(* IEC 61131-3 sources: verifaps-lib/share/PPU.stold (part 6) *)

(* ---- Scenario13_Final.xml.st ---- *)
TYPE
    Crane_states_t : (Crane_Go_Up , Crane_Go_Up_White , Crane_Init , Crane_Init_2 , Crane_Lift_At_Stamp , Crane_Lift_At_Stamp2 , Crane_Lift_Conveyor , Crane_Lift_Conveyor2 , Crane_Lift_Conveyor_Black , Crane_Lift_Magazin , Crane_Lift_Magazin_Metallic , Crane_Lift_Magazin_White , Crane_Lift_NOT_Metallic_Black , Crane_Lower , Crane_On_Conveyor , Crane_On_Conveyor_Metallic , Crane_On_Conveyor_Metallic2 , Crane_On_Conveyor_Not_Metallica_Black , Crane_On_Stamp_Metallic , Crane_On_Stamp_Metallic2 , Crane_On_Stamp_Metallic2_Lower , Crane_On_Stamp_Stop_Black , Crane_On_Stamp_White , Crane_Turn_Left_Back_To_Stamp , Crane_Turn_Left_From_Stamp , Crane_Turn_Left_Metallic , Crane_Turn_Left_Metallic2 , Crane_Turn_Left_NOT_Metallic , Crane_Turn_Left_NOT_Metallic_Black , Crane_Turn_Left_White , Crane_Turn_Right_From_Stamp , Init , Interstep , Interstep_2 , Interstep_3 , Interstep_4 , Lower_Crane , Magazin_Stop , Magazin_Stop_Black , Magazin_Stop_Final , No_Workpiece_ready , Reset_interconnect , Stamp_Pressure_Profile_Set_Metallic , Stamp_Pressure_Profile_Set_White , Start_Crane , Step0 , Step2 , Step3 , Step4 , Suck_At_Stamp , Suck_At_Stamp2 , TimeDelay , Turn_Right , Turn_Right_Black , Turn_Right_Final , pause , release , release2 , release_Black , release_Workpiece , release_Workpiece_White);
    Magazin_states_t : (Green_Lamp , Init , Interstep , Magazin_Init , Magazin_Init_2 , Slider_Move_Back , Start_Magazin , Step0 , Step1 , convey);
    Conveyor_states_t : (Conveyor_Init , Conveyor_Stop_Empty_Magazin , Conveyor_Towards_Stacker , Conveyor_init_2 , Conveyor_pause , Green_Lamp , Init , Interstep , Runtime_Conveyor , Start_Conveyor , Step0);
    Stamp_states_t : (Green_Lamp , Init , Interstep , Intertsep_2 , StampProcess , StampSliderBack , StampSliderForward , Stamp_Init_1 , Stamp_Init_2 , Stamp_Init_3 , Stamp_Init_4 , Start_Stamp , Step0 , Step1 , Step2);
    Pusher_states_t : (Check_For_Black , Check_For_Metal , Check_For_White , First_Slide_Timer_Black , First_Slide_Timer_Metal , First_Slide_Timer_White , First_Slide_black_workpieces , First_Slide_metal_workpieces , First_Slide_white_workpieces , Init , Interstep , Interstep_2 , PusherY1_Move_In_Black , PusherY1_Move_In_Metal , PusherY1_Move_In_White , PusherY1_Move_Out_Black , PusherY1_Move_Out_Metal , PusherY1_Move_Out_White , PusherY2_Move_In_Black , PusherY2_Move_In_Metal , PusherY2_Move_In_White , PusherY2_Move_Out_Black , PusherY2_Move_Out_Metal , PusherY2_Move_Out_White , Reset_interconnect3 , Reset_interconnect_Slide1_Black , Reset_interconnect_Slide1_Metal , Reset_interconnect_Slide1_White , Reset_interconnect_Slide2_Black , Reset_interconnect_Slide2_Metal , Reset_interconnect_Slide2_White , Reset_interconnect_Slide3_Metal , Reset_interconnect_Slide3_White , Second_Slide_Timer_Black , Second_Slide_Timer_Metal , Second_Slide_Timer_White , Second_Slide_black_workpieces , Second_Slide_metal_workpieces , Second_Slide_white_workpieces , Second_Test_For_Metal , Second_Test_For_White , Third_Slide_black_workpieces , Third_Slide_metal_workpieces , Third_Slide_white_workpieces , Wait_Black , Wait_Metal , Wait_White , Wait_Y1_Black , Wait_Y1_Metal , Wait_Y1_White , Wait_Y2_Black , Wait_Y2_Metal , Wait_Y2_White);
END_TYPE

FUNCTION_BLOCK Crane
    VAR_INPUT  AnalogCranePosition : INT; END_VAR {*Irwxp*}
    VAR_OUTPUT  AnalogCranePressure : INT; END_VAR {*Orwxp*}
    VAR_INPUT  CraneDown : BOOL; END_VAR {*Irwxp*}
    VAR_OUTPUT  CraneLower : BOOL; END_VAR {*Orwxp*}
    VAR_INPUT  CraneSucked : BOOL; END_VAR {*Irwxp*}
    VAR_OUTPUT  CraneTurnClockwise : BOOL; END_VAR {*Orwxp*}
    VAR_OUTPUT  CraneTurnCounterclockwise : BOOL; END_VAR {*Orwxp*}
    VAR_INPUT  CraneUp : BOOL; END_VAR {*Irwxp*}
    VAR  Duration1 : TIME := TIME#1.0s500.0ms; END_VAR {*Lrwxp*}
    VAR_INPUT  MagazinCapacitiveSensor : BOOL; END_VAR {*Irwxp*}
    VAR_INPUT  MagazinOpticalSensor : BOOL; END_VAR {*Irwxp*}
    VAR_OUTPUT  MagazinSlider : BOOL; END_VAR {*Orwxp*}
    VAR_OUTPUT  MagazinVacuumOff : BOOL; END_VAR {*Orwxp*}
    VAR_OUTPUT  MagazinVacuumOn : BOOL; END_VAR {*Orwxp*}
    VAR  SFCInit : BOOL; END_VAR {*Lrwxp*}
    VAR_INPUT  SFCReset : BOOL; END_VAR {*Irwxp*}
    VAR_INPUT  SliderMovedOut : BOOL; END_VAR {*Irwxp*}
    VAR_INPUT  SliderNotMovedOut : BOOL; END_VAR {*Irwxp*}
    VAR_INPUT  StampLowered : BOOL; END_VAR {*Irwxp*}
    VAR_INPUT  StampSliderFilled : BOOL; END_VAR {*Irwxp*}
    VAR_INPUT  StampSliderSensorMovedOut : BOOL; END_VAR {*Irwxp*}
    VAR_INPUT  StartButtonMagazin : BOOL; END_VAR {*Irwxp*}
    VAR_OUTPUT  StartCommandCrane : BOOL; END_VAR {*Orwxp*}
    VAR_INPUT  StartVar : BOOL; END_VAR {*Irwxp*}
    VAR  TimeDelay_Timer : TON; END_VAR {*Lrwxp*}
    VAR  TimeDelay_Timer_Duration : TIME := TIME#50.0ms; END_VAR {*Lrwxp*}
    VAR  TimeDelay_Timer_interconnect : BOOL; END_VAR {*Lrwxp*}
    VAR  Timer1 : TON; END_VAR {*Lrwxp*}
    VAR_INPUT  WorkpieceReady : BOOL; END_VAR {*Irwxp*}
    VAR  _state : Crane_states_t; END_VAR {*Lrwxp*}
    VAR  _transit : BOOL; END_VAR {*Lrwxp*}
    VAR  actualtime1 : TIME; END_VAR {*Lrwxp*}
    VAR  interconnect : BOOL; END_VAR {*Lrwxp*}
    VAR  interconnectCraneStartCommand : BOOL; END_VAR {*Lrwxp*}

    CASE _state OF
        Crane_states_t#Crane_Go_Up:
            {* begin(State) *}
            {* begin(onEntry) *}
            _transit := FALSE;
            {* end(onEntry) *}
            {* begin(onActive) *}
            CraneLower := FALSE;
            {* end(onActive) *}
            {* begin(transition) *}
            IF CraneUp THEN
                _transit := TRUE;
                _state := Crane_states_t#Step3;
            END_IF;
            {* end(transition) *}
            {* begin(onExit) *}
            {* end(onExit) *}
            {* end(State) *}

        Crane_states_t#Crane_Go_Up_White:
            {* begin(State) *}
            {* begin(onEntry) *}
            _transit := FALSE;
            {* end(onEntry) *}
            {* begin(onActive) *}
            CraneLower := FALSE;
            {* end(onActive) *}
            {* begin(transition) *}
            IF CraneUp THEN
                _transit := TRUE;
                _state := Crane_states_t#Step3;
            END_IF;
            {* end(transition) *}
            {* begin(onExit) *}
            {* end(onExit) *}
            {* end(State) *}

        Crane_states_t#Crane_Init:
            {* begin(State) *}
            {* begin(onEntry) *}
            _transit := FALSE;
            {* end(onEntry) *}
            {* begin(onActive) *}
            CraneLower := TRUE;
            interconnectCraneStartCommand := FALSE;
            AnalogCranePressure := INT#6000;
            {* end(onActive) *}
            {* begin(transition) *}
            IF CraneDown THEN
                _transit := TRUE;
                _state := Crane_states_t#Crane_Init_2;
            END_IF;
            {* end(transition) *}
            {* begin(onExit) *}
            {* end(onExit) *}
            {* end(State) *}

        Crane_states_t#Crane_Init_2:
            {* begin(State) *}
            {* begin(onEntry) *}
            _transit := FALSE;
            {* end(onEntry) *}
            {* begin(onActive) *}
            CraneLower := FALSE;
            {* end(onActive) *}
            {* begin(transition) *}
            IF CraneUp THEN
                _transit := TRUE;
                _state := Crane_states_t#Interstep;
            END_IF;
            {* end(transition) *}
            {* begin(onExit) *}
            {* end(onExit) *}
            {* end(State) *}

        Crane_states_t#Crane_Lift_At_Stamp:
            {* begin(State) *}
            {* begin(onEntry) *}
            _transit := FALSE;
            {* end(onEntry) *}
            {* begin(onActive) *}
            CraneLower := FALSE;
            {* end(onActive) *}
            {* begin(transition) *}
            IF CraneUp THEN
                _transit := TRUE;
                _state := Crane_states_t#Crane_Turn_Left_From_Stamp;
            END_IF;
            {* end(transition) *}
            {* begin(onExit) *}
            {* end(onExit) *}
            {* end(State) *}

        Crane_states_t#Crane_Lift_At_Stamp2:
            {* begin(State) *}
            {* begin(onEntry) *}
            _transit := FALSE;
            {* end(onEntry) *}
            {* begin(onActive) *}
            CraneLower := FALSE;
            AnalogCranePressure := INT#0;
            {* end(onActive) *}
            {* begin(transition) *}
            IF CraneUp THEN
                _transit := TRUE;
                _state := Crane_states_t#Crane_Turn_Right_From_Stamp;
            END_IF;
            {* end(transition) *}
            {* begin(onExit) *}
            {* end(onExit) *}
            {* end(State) *}

        Crane_states_t#Crane_Lift_Conveyor:
            {* begin(State) *}
            {* begin(onEntry) *}
            _transit := FALSE;
            {* end(onEntry) *}
            {* begin(onActive) *}
            CraneLower := FALSE;
            {* end(onActive) *}
            {* begin(transition) *}
            IF TRUE THEN
                _transit := TRUE;
                _state := Crane_states_t#Interstep;
            END_IF;
            {* end(transition) *}
            {* begin(onExit) *}
            {* end(onExit) *}
            {* end(State) *}

        Crane_states_t#Crane_Lift_Conveyor2:
            {* begin(State) *}
            {* begin(onEntry) *}
            _transit := FALSE;
            {* end(onEntry) *}
            {* begin(onActive) *}
            CraneLower := FALSE;
            {* end(onActive) *}
            {* begin(transition) *}
            IF TRUE THEN
                _transit := TRUE;
                _state := Crane_states_t#Interstep;
            END_IF;
            {* end(transition) *}
            {* begin(onExit) *}
            {* end(onExit) *}
            {* end(State) *}

        Crane_states_t#Crane_Lift_Conveyor_Black:
            {* begin(State) *}
            {* begin(onEntry) *}
            _transit := FALSE;
            {* end(onEntry) *}
            {* begin(onActive) *}
            CraneLower := FALSE;
            {* end(onActive) *}
            {* begin(transition) *}
            IF CraneUp THEN
                _transit := TRUE;
                _state := Crane_states_t#Crane_Turn_Left_Back_To_Stamp;
            END_IF;
            {* end(transition) *}
            {* begin(onExit) *}
            {* end(onExit) *}
            {* end(State) *}

        Crane_states_t#Crane_Lift_Magazin:
            {* begin(State) *}
            {* begin(onEntry) *}
            _transit := FALSE;
            {* end(onEntry) *}
            {* begin(onActive) *}
            CraneLower := FALSE;
            {* end(onActive) *}
            {* begin(transition) *}
            IF CraneUp THEN
                _transit := TRUE;
                _state := Crane_states_t#Crane_Turn_Left_NOT_Metallic;
            END_IF;
            {* end(transition) *}
            {* begin(onExit) *}
            {* end(onExit) *}
            {* end(State) *}

        Crane_states_t#Crane_Lift_Magazin_Metallic:
            {* begin(State) *}
            {* begin(onEntry) *}
            _transit := FALSE;
            {* end(onEntry) *}
            {* begin(onActive) *}
            CraneLower := FALSE;
            {* end(onActive) *}
            {* begin(transition) *}
            IF CraneUp THEN
                _transit := TRUE;
                _state := Crane_states_t#Crane_Turn_Left_Metallic;
            END_IF;
            {* end(transition) *}
            {* begin(onExit) *}
            {* end(onExit) *}
            {* end(State) *}

        Crane_states_t#Crane_Lift_Magazin_White:
            {* begin(State) *}
            {* begin(onEntry) *}
            _transit := FALSE;
            {* end(onEntry) *}
            {* begin(onActive) *}
            CraneLower := FALSE;
            {* end(onActive) *}
            {* begin(transition) *}
            IF CraneUp THEN
                _transit := TRUE;
                _state := Crane_states_t#Crane_Turn_Left_White;
            END_IF;
            {* end(transition) *}
            {* begin(onExit) *}
            {* end(onExit) *}
            {* end(State) *}

        Crane_states_t#Crane_Lift_NOT_Metallic_Black:
            {* begin(State) *}
            {* begin(onEntry) *}
            _transit := FALSE;
            {* end(onEntry) *}
            {* begin(onActive) *}
            CraneLower := FALSE;
            {* end(onActive) *}
            {* begin(transition) *}
            IF CraneUp THEN
                _transit := TRUE;
                _state := Crane_states_t#Crane_Turn_Left_NOT_Metallic_Black;
            END_IF;
            {* end(transition) *}
            {* begin(onExit) *}
            {* end(onExit) *}
            {* end(State) *}

        Crane_states_t#Crane_Lower:
            {* begin(State) *}
            {* begin(onEntry) *}
            _transit := FALSE;
            {* end(onEntry) *}
            {* begin(onActive) *}
            MagazinVacuumOn := TRUE;
            MagazinVacuumOff := FALSE;
            CraneLower := TRUE;
            AnalogCranePressure := INT#0;
            {* end(onActive) *}
            {* begin(transition) *}
            IF CraneSucked THEN
                _transit := TRUE;
                _state := Crane_states_t#Step0;
            END_IF;
            {* end(transition) *}
            {* begin(onExit) *}
            {* end(onExit) *}
            {* end(State) *}

        Crane_states_t#Crane_On_Conveyor:
            {* begin(State) *}
            {* begin(onEntry) *}
            _transit := FALSE;
            {* end(onEntry) *}
            {* begin(onActive) *}
            CraneTurnCounterclockwise := FALSE;
            CraneTurnClockwise := FALSE;
            CraneLower := TRUE;
            {* end(onActive) *}
            {* begin(transition) *}
            IF CraneDown THEN
                _transit := TRUE;
                _state := Crane_states_t#release;
            END_IF;
            {* end(transition) *}
            {* begin(onExit) *}
            {* end(onExit) *}
            {* end(State) *}

        Crane_states_t#Crane_On_Conveyor_Metallic:
            {* begin(State) *}
            {* begin(onEntry) *}
            _transit := FALSE;
            {* end(onEntry) *}
            {* begin(onActive) *}
            CraneTurnCounterclockwise := FALSE;
            CraneTurnClockwise := FALSE;
            CraneLower := TRUE;
            {* end(onActive) *}
            {* begin(transition) *}
            IF CraneDown THEN
                _transit := TRUE;
                _state := Crane_states_t#release;
            END_IF;
            {* end(transition) *}
            {* begin(onExit) *}
            {* end(onExit) *}
            {* end(State) *}

        Crane_states_t#Crane_On_Conveyor_Metallic2:
            {* begin(State) *}
            {* begin(onEntry) *}
            _transit := FALSE;
            {* end(onEntry) *}
            {* begin(onActive) *}
            CraneTurnCounterclockwise := FALSE;
            CraneTurnClockwise := FALSE;
            CraneLower := TRUE;
            {* end(onActive) *}
            {* begin(transition) *}
            IF CraneDown THEN
                _transit := TRUE;
                _state := Crane_states_t#release2;
            END_IF;
            {* end(transition) *}
            {* begin(onExit) *}
            {* end(onExit) *}
            {* end(State) *}

        Crane_states_t#Crane_On_Conveyor_Not_Metallica_Black:
            {* begin(State) *}
            {* begin(onEntry) *}
            _transit := FALSE;
            {* end(onEntry) *}
            {* begin(onActive) *}
            CraneTurnCounterclockwise := FALSE;
            CraneTurnClockwise := FALSE;
            CraneLower := TRUE;
            {* end(onActive) *}
            {* begin(transition) *}
            IF CraneDown THEN
                _transit := TRUE;
                _state := Crane_states_t#release_Black;
            END_IF;
            {* end(transition) *}
            {* begin(onExit) *}
            {* end(onExit) *}
            {* end(State) *}

        Crane_states_t#Crane_On_Stamp_Metallic:
            {* begin(State) *}
            {* begin(onEntry) *}
            _transit := FALSE;
            {* end(onEntry) *}
            {* begin(onActive) *}
            CraneTurnCounterclockwise := FALSE;
            CraneTurnClockwise := FALSE;
            CraneLower := TRUE;
            {* end(onActive) *}
            {* begin(transition) *}
            IF CraneDown THEN
                _transit := TRUE;
                _state := Crane_states_t#release_Workpiece;
            END_IF;
            {* end(transition) *}
            {* begin(onExit) *}
            {* end(onExit) *}
            {* end(State) *}

        Crane_states_t#Crane_On_Stamp_Metallic2:
            {* begin(State) *}
            {* begin(onEntry) *}
            _transit := FALSE;
            {* end(onEntry) *}
            {* begin(onActive) *}
            CraneTurnCounterclockwise := FALSE;
            CraneTurnClockwise := FALSE;
            {* end(onActive) *}
            {* begin(transition) *}
            IF StampLowered THEN
                _transit := TRUE;
                _state := Crane_states_t#Interstep_4;
            END_IF;
            {* end(transition) *}
            {* begin(onExit) *}
            {* end(onExit) *}
            {* end(State) *}

        Crane_states_t#Crane_On_Stamp_Metallic2_Lower:
            {* begin(State) *}
            {* begin(onEntry) *}
            _transit := FALSE;
            {* end(onEntry) *}
            {* begin(onActive) *}
            CraneLower := TRUE;
            {* end(onActive) *}
            {* begin(transition) *}
            IF CraneDown THEN
                _transit := TRUE;
                _state := Crane_states_t#Suck_At_Stamp2;
            END_IF;
            {* end(transition) *}
            {* begin(onExit) *}
            {* end(onExit) *}
            {* end(State) *}

        Crane_states_t#Crane_On_Stamp_Stop_Black:
            {* begin(State) *}
            {* begin(onEntry) *}
            _transit := FALSE;
            {* end(onEntry) *}
            {* begin(onActive) *}
            CraneTurnClockwise := FALSE;
            CraneTurnCounterclockwise := FALSE;
            {* end(onActive) *}
            {* begin(transition) *}
            IF TRUE THEN
                _transit := TRUE;
                _state := Crane_states_t#Reset_interconnect;
            END_IF;
            {* end(transition) *}
            {* begin(onExit) *}
            {* end(onExit) *}
            {* end(State) *}

        Crane_states_t#Crane_On_Stamp_White:
            {* begin(State) *}
            {* begin(onEntry) *}
            _transit := FALSE;
            {* end(onEntry) *}
            {* begin(onActive) *}
            CraneTurnCounterclockwise := FALSE;
            CraneTurnClockwise := FALSE;
            CraneLower := TRUE;
            {* end(onActive) *}
            {* begin(transition) *}
            IF CraneDown THEN
                _transit := TRUE;
                _state := Crane_states_t#release_Workpiece_White;
            END_IF;
            {* end(transition) *}
            {* begin(onExit) *}
            {* end(onExit) *}
            {* end(State) *}

        Crane_states_t#Crane_Turn_Left_Back_To_Stamp:
            {* begin(State) *}
            {* begin(onEntry) *}
            _transit := FALSE;
            {* end(onEntry) *}
            {* begin(onActive) *}
            CraneTurnCounterclockwise := TRUE;
            CraneTurnClockwise := FALSE;
            {* end(onActive) *}
            {* begin(transition) *}
            IF ((AnalogCranePosition > INT#8160) AND (AnalogCranePosition < INT#8260)) THEN
                _transit := TRUE;
                _state := Crane_states_t#Crane_On_Stamp_Stop_Black;
            END_IF;
            {* end(transition) *}
            {* begin(onExit) *}
            {* end(onExit) *}
            {* end(State) *}

        Crane_states_t#Crane_Turn_Left_From_Stamp:
            {* begin(State) *}
            {* begin(onEntry) *}
            _transit := FALSE;
            {* end(onEntry) *}
            {* begin(onActive) *}
            CraneTurnClockwise := TRUE;
            CraneTurnCounterclockwise := FALSE;
            {* end(onActive) *}
            {* begin(transition) *}
            IF ((AnalogCranePosition > INT#16060) AND (AnalogCranePosition < INT#16160)) THEN
                _transit := TRUE;
                _state := Crane_states_t#Crane_On_Conveyor_Metallic;
            END_IF;
            {* end(transition) *}
            {* begin(onExit) *}
            {* end(onExit) *}
            {* end(State) *}

        Crane_states_t#Crane_Turn_Left_Metallic:
            {* begin(State) *}
            {* begin(onEntry) *}
            _transit := FALSE;
            {* end(onEntry) *}
            {* begin(onActive) *}
            CraneTurnCounterclockwise := TRUE;
            CraneTurnClockwise := FALSE;
            {* end(onActive) *}
            {* begin(transition) *}
            IF ((AnalogCranePosition > INT#8160) AND (AnalogCranePosition < INT#8260)) THEN
                _transit := TRUE;
                _state := Crane_states_t#Crane_On_Stamp_Metallic;
            END_IF;
            {* end(transition) *}
            {* begin(onExit) *}
            {* end(onExit) *}
            {* end(State) *}

        Crane_states_t#Crane_Turn_Left_Metallic2:
            {* begin(State) *}
            {* begin(onEntry) *}
            _transit := FALSE;
            {* end(onEntry) *}
            {* begin(onActive) *}
            CraneTurnCounterclockwise := TRUE;
            CraneTurnClockwise := FALSE;
            {* end(onActive) *}
            {* begin(transition) *}
            IF ((AnalogCranePosition > INT#8160) AND (AnalogCranePosition < INT#8260)) THEN
                _transit := TRUE;
                _state := Crane_states_t#Crane_On_Stamp_Metallic2;
            END_IF;
            {* end(transition) *}
            {* begin(onExit) *}
            {* end(onExit) *}
            {* end(State) *}

        Crane_states_t#Crane_Turn_Left_NOT_Metallic:
            {* begin(State) *}
            {* begin(onEntry) *}
            _transit := FALSE;
            {* end(onEntry) *}
            {* begin(onActive) *}
            CraneTurnCounterclockwise := TRUE;
            CraneTurnClockwise := FALSE;
            {* end(onActive) *}
            {* begin(transition) *}
            IF ((AnalogCranePosition > INT#16160) AND (AnalogCranePosition < INT#16260)) THEN
                _transit := TRUE;
                _state := Crane_states_t#Crane_On_Conveyor;
            END_IF;
            {* end(transition) *}
            {* begin(onExit) *}
            {* end(onExit) *}
            {* end(State) *}

        Crane_states_t#Crane_Turn_Left_NOT_Metallic_Black:
            {* begin(State) *}
            {* begin(onEntry) *}
            _transit := FALSE;
            {* end(onEntry) *}
            {* begin(onActive) *}
            CraneTurnCounterclockwise := TRUE;
            CraneTurnClockwise := FALSE;
            {* end(onActive) *}
            {* begin(transition) *}
            IF ((AnalogCranePosition > INT#16160) AND (AnalogCranePosition < INT#16260)) THEN
                _transit := TRUE;
                _state := Crane_states_t#Crane_On_Conveyor_Not_Metallica_Black;
            END_IF;
            {* end(transition) *}
            {* begin(onExit) *}
            {* end(onExit) *}
            {* end(State) *}

        Crane_states_t#Crane_Turn_Left_White:
            {* begin(State) *}
            {* begin(onEntry) *}
            _transit := FALSE;
            {* end(onEntry) *}
            {* begin(onActive) *}
            CraneTurnCounterclockwise := TRUE;
            CraneTurnClockwise := FALSE;
            {* end(onActive) *}
            {* begin(transition) *}
            IF ((AnalogCranePosition > INT#8160) AND (AnalogCranePosition < INT#8260)) THEN
                _transit := TRUE;
                _state := Crane_states_t#Crane_On_Stamp_White;
            END_IF;
            {* end(transition) *}
            {* begin(onExit) *}
            {* end(onExit) *}
            {* end(State) *}

        Crane_states_t#Crane_Turn_Right_From_Stamp:
            {* begin(State) *}
            {* begin(onEntry) *}
            _transit := FALSE;
            {* end(onEntry) *}
            {* begin(onActive) *}
            CraneTurnClockwise := TRUE;
            CraneTurnCounterclockwise := FALSE;
            {* end(onActive) *}
            {* begin(transition) *}
            IF ((AnalogCranePosition > INT#16160) AND (AnalogCranePosition < INT#16260)) THEN
                _transit := TRUE;
                _state := Crane_states_t#Crane_On_Conveyor_Metallic2;
            END_IF;
            {* end(transition) *}
            {* begin(onExit) *}
            {* end(onExit) *}
            {* end(State) *}

        Crane_states_t#Init:
            {* begin(State) *}
            {* begin(onEntry) *}
            _transit := FALSE;
            {* end(onEntry) *}
            {* begin(onActive) *}
            {* end(onActive) *}
            {* begin(transition) *}
            IF TRUE THEN
                _transit := TRUE;
                _state := Crane_states_t#Start_Crane;
            END_IF;
            {* end(transition) *}
            {* begin(onExit) *}
            {* end(onExit) *}
            {* end(State) *}

        Crane_states_t#Interstep:
            {* begin(State) *}
            {* begin(onEntry) *}
            _transit := FALSE;
            {* end(onEntry) *}
            {* begin(onActive) *}
            StartCommandCrane := TRUE;
            {* end(onActive) *}
            {* begin(transition) *}
            IF StartVar THEN
                _transit := TRUE;
                _state := Crane_states_t#Interstep_2;
            END_IF;
            {* end(transition) *}
            {* begin(onExit) *}
            {* end(onExit) *}
            {* end(State) *}

        Crane_states_t#Interstep_2:
            {* begin(State) *}
            {* begin(onEntry) *}
            _transit := FALSE;
            {* end(onEntry) *}
            {* begin(onActive) *}
            {* end(onActive) *}
            {* begin(transition) *}
            IF SliderMovedOut THEN
                _transit := TRUE;
                _state := Crane_states_t#TimeDelay;
            END_IF;
            {* end(transition) *}
            {* begin(onExit) *}
            {* end(onExit) *}
            {* end(State) *}

        Crane_states_t#Interstep_3:
            {* begin(State) *}
            {* begin(onEntry) *}
            _transit := FALSE;
            {* end(onEntry) *}
            {* begin(onActive) *}
            {* end(onActive) *}
            {* begin(transition) *}
            IF NOT WorkpieceReady THEN
                _transit := TRUE;
                _state := Crane_states_t#No_Workpiece_ready;
            ELSEIF WorkpieceReady THEN
                _transit := TRUE;
                _state := Crane_states_t#Turn_Right;
            END_IF;
            {* end(transition) *}
            {* begin(onExit) *}
            {* end(onExit) *}
            {* end(State) *}

        Crane_states_t#Interstep_4:
            {* begin(State) *}
            {* begin(onEntry) *}
            _transit := FALSE;
            {* end(onEntry) *}
            {* begin(onActive) *}
            {* end(onActive) *}
            {* begin(transition) *}
            IF StampSliderSensorMovedOut THEN
                _transit := TRUE;
                _state := Crane_states_t#Crane_On_Stamp_Metallic2_Lower;
            END_IF;
            {* end(transition) *}
            {* begin(onExit) *}
            {* end(onExit) *}
            {* end(State) *}

        Crane_states_t#Lower_Crane:
            {* begin(State) *}
            {* begin(onEntry) *}
            _transit := FALSE;
            {* end(onEntry) *}
            {* begin(onActive) *}
            CraneLower := TRUE;
            {* end(onActive) *}
            {* begin(transition) *}
            IF CraneDown THEN
                _transit := TRUE;
                _state := Crane_states_t#Suck_At_Stamp;
            END_IF;
            {* end(transition) *}
            {* begin(onExit) *}
            {* end(onExit) *}
            {* end(State) *}

        Crane_states_t#Magazin_Stop:
            {* begin(State) *}
            {* begin(onEntry) *}
            _transit := FALSE;
            {* end(onEntry) *}
            {* begin(onActive) *}
            CraneTurnClockwise := FALSE;
            CraneTurnCounterclockwise := FALSE;
            {* end(onActive) *}
            {* begin(transition) *}
            IF TRUE THEN
                _transit := TRUE;
                _state := Crane_states_t#Crane_Lower;
            END_IF;
            {* end(transition) *}
            {* begin(onExit) *}
            {* end(onExit) *}
            {* end(State) *}

        Crane_states_t#Magazin_Stop_Black:
            {* begin(State) *}
            {* begin(onEntry) *}
            _transit := FALSE;
            {* end(onEntry) *}
            {* begin(onActive) *}
            CraneTurnClockwise := FALSE;
            CraneTurnCounterclockwise := FALSE;
            MagazinVacuumOn := TRUE;
            MagazinVacuumOff := FALSE;
            CraneLower := TRUE;
            {* end(onActive) *}
            {* begin(transition) *}
            IF CraneSucked THEN
                _transit := TRUE;
                _state := Crane_states_t#Crane_Lift_NOT_Metallic_Black;
            END_IF;
            {* end(transition) *}
            {* begin(onExit) *}
            {* end(onExit) *}
            {* end(State) *}

        Crane_states_t#Magazin_Stop_Final:
            {* begin(State) *}
            {* begin(onEntry) *}
            _transit := FALSE;
            {* end(onEntry) *}
            {* begin(onActive) *}
            CraneTurnClockwise := FALSE;
            CraneTurnCounterclockwise := FALSE;
            {* end(onActive) *}
            {* begin(transition) *}
            IF TRUE THEN
                _transit := TRUE;
                _state := Crane_states_t#Start_Crane;
            END_IF;
            {* end(transition) *}
            {* begin(onExit) *}
            {* end(onExit) *}
            {* end(State) *}

        Crane_states_t#No_Workpiece_ready:
            {* begin(State) *}
            {* begin(onEntry) *}
            _transit := FALSE;
            {* end(onEntry) *}
            {* begin(onActive) *}
            MagazinVacuumOn := FALSE;
            MagazinVacuumOff := FALSE;
            CraneLower := FALSE;
            {* end(onActive) *}
            {* begin(transition) *}
            IF StampSliderFilled THEN
                _transit := TRUE;
                _state := Crane_states_t#Crane_Turn_Left_Metallic2;
            ELSEIF NOT StampSliderFilled THEN
                _transit := TRUE;
                _state := Crane_states_t#Turn_Right_Final;
            END_IF;
            {* end(transition) *}
            {* begin(onExit) *}
            {* end(onExit) *}
            {* end(State) *}

        Crane_states_t#Reset_interconnect:
            {* begin(State) *}
            {* begin(onEntry) *}
            _transit := FALSE;
            {* end(onEntry) *}
            {* begin(onActive) *}
            interconnect := FALSE;
            Timer1(IN := FALSE, PT := TIME#1.0ms);
            {* end(onActive) *}
            {* begin(transition) *}
            IF SliderMovedOut THEN
                _transit := TRUE;
                _state := Crane_states_t#Lower_Crane;
            END_IF;
            {* end(transition) *}
            {* begin(onExit) *}
            {* end(onExit) *}
            {* end(State) *}

        Crane_states_t#Stamp_Pressure_Profile_Set_Metallic:
            {* begin(State) *}
            {* begin(onEntry) *}
            _transit := FALSE;
            {* end(onEntry) *}
            {* begin(onActive) *}
            AnalogCranePressure := INT#7000;
            {* end(onActive) *}
            {* begin(transition) *}
            IF TRUE THEN
                _transit := TRUE;
                _state := Crane_states_t#Crane_Lift_Magazin_Metallic;
            END_IF;
            {* end(transition) *}
            {* begin(onExit) *}
            {* end(onExit) *}
            {* end(State) *}

        Crane_states_t#Stamp_Pressure_Profile_Set_White:
            {* begin(State) *}
            {* begin(onEntry) *}
            _transit := FALSE;
            {* end(onEntry) *}
            {* begin(onActive) *}
            AnalogCranePressure := INT#6000;
            {* end(onActive) *}
            {* begin(transition) *}
            IF TRUE THEN
                _transit := TRUE;
                _state := Crane_states_t#Crane_Lift_Magazin_White;
            END_IF;
            {* end(transition) *}
            {* begin(onExit) *}
            {* end(onExit) *}
            {* end(State) *}

        Crane_states_t#Start_Crane:
            {* begin(State) *}
            {* begin(onEntry) *}
            _transit := FALSE;
            {* end(onEntry) *}
            {* begin(onActive) *}
            CraneLower := FALSE;
            MagazinVacuumOff := FALSE;
            MagazinVacuumOn := FALSE;
            CraneTurnCounterclockwise := FALSE;
            CraneTurnClockwise := FALSE;
            AnalogCranePressure := INT#0;
            StartVar := FALSE;
            StartCommandCrane := FALSE;
            IF (StartButtonMagazin = TRUE) THEN
                interconnectCraneStartCommand := TRUE;
            END_IF;
            {* end(onActive) *}
            {* begin(transition) *}
            IF interconnectCraneStartCommand THEN
                _transit := TRUE;
                _state := Crane_states_t#Crane_Init;
            END_IF;
            {* end(transition) *}
            {* begin(onExit) *}
            {* end(onExit) *}
            {* end(State) *}

        Crane_states_t#Step0:
            {* begin(State) *}
            {* begin(onEntry) *}
            _transit := FALSE;
            {* end(onEntry) *}
            {* begin(onActive) *}
            {* end(onActive) *}
            {* begin(transition) *}
            IF (MagazinCapacitiveSensor AND MagazinOpticalSensor) THEN
                _transit := TRUE;
                _state := Crane_states_t#Stamp_Pressure_Profile_Set_Metallic;
            ELSEIF (NOT MagazinCapacitiveSensor AND MagazinOpticalSensor) THEN
                _transit := TRUE;
                _state := Crane_states_t#Stamp_Pressure_Profile_Set_White;
            ELSEIF (NOT MagazinCapacitiveSensor AND NOT MagazinOpticalSensor) THEN
                _transit := TRUE;
                _state := Crane_states_t#Crane_Lift_Magazin;
            END_IF;
            {* end(transition) *}
            {* begin(onExit) *}
            {* end(onExit) *}
            {* end(State) *}

        Crane_states_t#Step2:
            {* begin(State) *}
            {* begin(onEntry) *}
            _transit := FALSE;
            {* end(onEntry) *}
            {* begin(onActive) *}
            {* end(onActive) *}
            {* begin(transition) *}
            IF (MagazinCapacitiveSensor OR MagazinOpticalSensor) THEN
                _transit := TRUE;
                _state := Crane_states_t#pause;
            ELSEIF (NOT MagazinCapacitiveSensor AND NOT MagazinOpticalSensor) THEN
                _transit := TRUE;
                _state := Crane_states_t#Turn_Right_Black;
            END_IF;
            {* end(transition) *}
            {* begin(onExit) *}
            {* end(onExit) *}
            {* end(State) *}

        Crane_states_t#Step3:
            {* begin(State) *}
            {* begin(onEntry) *}
            _transit := FALSE;
            {* end(onEntry) *}
            {* begin(onActive) *}
            {* end(onActive) *}
            {* begin(transition) *}
            IF NOT WorkpieceReady THEN
                _transit := TRUE;
                _state := Crane_states_t#Step4;
            ELSEIF WorkpieceReady THEN
                _transit := TRUE;
                _state := Crane_states_t#Step2;
            END_IF;
            {* end(transition) *}
            {* begin(onExit) *}
            {* end(onExit) *}
            {* end(State) *}

        Crane_states_t#Step4:
            {* begin(State) *}
            {* begin(onEntry) *}
            _transit := FALSE;
            {* end(onEntry) *}
            {* begin(onActive) *}
            {* end(onActive) *}
            {* begin(transition) *}
            IF TRUE THEN
                _transit := TRUE;
                _state := Crane_states_t#Interstep;
            END_IF;
            {* end(transition) *}
            {* begin(onExit) *}
            {* end(onExit) *}
            {* end(State) *}

        Crane_states_t#Suck_At_Stamp:
            {* begin(State) *}
            {* begin(onEntry) *}
            _transit := FALSE;
            {* end(onEntry) *}
            {* begin(onActive) *}
            MagazinVacuumOn := TRUE;
            MagazinVacuumOff := FALSE;
            {* end(onActive) *}
            {* begin(transition) *}
            IF CraneSucked THEN
                _transit := TRUE;
                _state := Crane_states_t#Crane_Lift_At_Stamp;
            END_IF;
            {* end(transition) *}
            {* begin(onExit) *}
            {* end(onExit) *}
            {* end(State) *}

        Crane_states_t#Suck_At_Stamp2:
            {* begin(State) *}
            {* begin(onEntry) *}
            _transit := FALSE;
            {* end(onEntry) *}
            {* begin(onActive) *}
            MagazinVacuumOn := TRUE;
            MagazinVacuumOff := FALSE;
            {* end(onActive) *}
            {* begin(transition) *}
            IF CraneSucked THEN
                _transit := TRUE;
                _state := Crane_states_t#Crane_Lift_At_Stamp2;
            END_IF;
            {* end(transition) *}
            {* begin(onExit) *}
            {* end(onExit) *}
            {* end(State) *}

        Crane_states_t#TimeDelay:
            {* begin(State) *}
            {* begin(onEntry) *}
            _transit := FALSE;
            {* end(onEntry) *}
            {* begin(onActive) *}
            TimeDelay_Timer(IN := TRUE, PT := TimeDelay_Timer_Duration);
            TimeDelay_Timer_interconnect := TimeDelay_Timer.Q;
            {* end(onActive) *}
            {* begin(transition) *}
            IF TimeDelay_Timer_interconnect THEN
                _transit := TRUE;
                _state := Crane_states_t#Interstep_3;
            END_IF;
            {* end(transition) *}
            {* begin(onExit) *}
            {* end(onExit) *}
            {* end(State) *}

        Crane_states_t#Turn_Right:
            {* begin(State) *}
            {* begin(onEntry) *}
            _transit := FALSE;
            {* end(onEntry) *}
            {* begin(onActive) *}
            CraneTurnClockwise := TRUE;
            CraneTurnCounterclockwise := FALSE;
            {* end(onActive) *}
            {* begin(transition) *}
            IF ((AnalogCranePosition > INT#24290) AND (AnalogCranePosition < INT#24390)) THEN
                _transit := TRUE;
                _state := Crane_states_t#Magazin_Stop;
            END_IF;
            {* end(transition) *}
            {* begin(onExit) *}
            {* end(onExit) *}
            {* end(State) *}

        Crane_states_t#Turn_Right_Black:
            {* begin(State) *}
            {* begin(onEntry) *}
            _transit := FALSE;
            {* end(onEntry) *}
            {* begin(onActive) *}
            CraneTurnClockwise := TRUE;
            CraneTurnCounterclockwise := FALSE;
            {* end(onActive) *}
            {* begin(transition) *}
            IF ((AnalogCranePosition > INT#24290) AND (AnalogCranePosition < INT#24390)) THEN
                _transit := TRUE;
                _state := Crane_states_t#Magazin_Stop_Black;
            END_IF;
            {* end(transition) *}
            {* begin(onExit) *}
            {* end(onExit) *}
            {* end(State) *}

        Crane_states_t#Turn_Right_Final:
            {* begin(State) *}
            {* begin(onEntry) *}
            _transit := FALSE;
            {* end(onEntry) *}
            {* begin(onActive) *}
            CraneTurnClockwise := TRUE;
            CraneTurnCounterclockwise := FALSE;
            AnalogCranePressure := INT#0;
            {* end(onActive) *}
            {* begin(transition) *}
            IF ((AnalogCranePosition > INT#24290) AND (AnalogCranePosition < INT#24390)) THEN
                _transit := TRUE;
                _state := Crane_states_t#Magazin_Stop_Final;
            END_IF;
            {* end(transition) *}
            {* begin(onExit) *}
            {* end(onExit) *}
            {* end(State) *}

        Crane_states_t#pause:
            {* begin(State) *}
            {* begin(onEntry) *}
            _transit := FALSE;
            {* end(onEntry) *}
            {* begin(onActive) *}
            Timer1(IN := CraneUp, PT := Duration1);
            interconnect := Timer1.Q;
            {* end(onActive) *}
            {* begin(transition) *}
            IF interconnect THEN
                _transit := TRUE;
                _state := Crane_states_t#Reset_interconnect;
            END_IF;
            {* end(transition) *}
            {* begin(onExit) *}
            {* end(onExit) *}
            {* end(State) *}

        Crane_states_t#release:
            {* begin(State) *}
            {* begin(onEntry) *}
            _transit := FALSE;
            {* end(onEntry) *}
            {* begin(onActive) *}
            MagazinVacuumOff := TRUE;
            MagazinVacuumOn := FALSE;
            {* end(onActive) *}
            {* begin(transition) *}
            IF TRUE THEN
                _transit := TRUE;
                _state := Crane_states_t#Crane_Lift_Conveyor;
            END_IF;
            {* end(transition) *}
            {* begin(onExit) *}
            {* end(onExit) *}
            {* end(State) *}

        Crane_states_t#release2:
            {* begin(State) *}
            {* begin(onEntry) *}
            _transit := FALSE;
            {* end(onEntry) *}
            {* begin(onActive) *}
            MagazinVacuumOff := TRUE;
            MagazinVacuumOn := FALSE;
            {* end(onActive) *}
            {* begin(transition) *}
            IF TRUE THEN
                _transit := TRUE;
                _state := Crane_states_t#Crane_Lift_Conveyor2;
            END_IF;
            {* end(transition) *}
            {* begin(onExit) *}
            {* end(onExit) *}
            {* end(State) *}

        Crane_states_t#release_Black:
            {* begin(State) *}
            {* begin(onEntry) *}
            _transit := FALSE;
            {* end(onEntry) *}
            {* begin(onActive) *}
            MagazinVacuumOn := FALSE;
            MagazinVacuumOff := TRUE;
            {* end(onActive) *}
            {* begin(transition) *}
            IF TRUE THEN
                _transit := TRUE;
                _state := Crane_states_t#Crane_Lift_Conveyor_Black;
            END_IF;
            {* end(transition) *}
            {* begin(onExit) *}
            {* end(onExit) *}
            {* end(State) *}

        Crane_states_t#release_Workpiece:
            {* begin(State) *}
            {* begin(onEntry) *}
            _transit := FALSE;
            {* end(onEntry) *}
            {* begin(onActive) *}
            MagazinVacuumOff := TRUE;
            MagazinVacuumOn := FALSE;
            {* end(onActive) *}
            {* begin(transition) *}
            IF TRUE THEN
                _transit := TRUE;
                _state := Crane_states_t#Crane_Go_Up;
            END_IF;
            {* end(transition) *}
            {* begin(onExit) *}
            {* end(onExit) *}
            {* end(State) *}

        Crane_states_t#release_Workpiece_White:
            {* begin(State) *}
            {* begin(onEntry) *}
            _transit := FALSE;
            {* end(onEntry) *}
            {* begin(onActive) *}
            MagazinVacuumOff := TRUE;
            MagazinVacuumOn := FALSE;
            {* end(onActive) *}
            {* begin(transition) *}
            IF TRUE THEN
                _transit := TRUE;
                _state := Crane_states_t#Crane_Go_Up_White;
            END_IF;
            {* end(transition) *}
            {* begin(onExit) *}
            {* end(onExit) *}
            {* end(State) *}

            END_CASE;
END_FUNCTION_BLOCK

FUNCTION_BLOCK Magazin
    VAR_INPUT  AnalogCranePosition : INT; END_VAR {*Irwxp*}
    VAR_INPUT  CraneDown : BOOL; END_VAR {*Irwxp*}
    VAR_OUTPUT  CraneLower : BOOL; END_VAR {*Orwxp*}
    VAR_INPUT  CraneOnConveyor : BOOL; END_VAR {*Irwxp*}
    VAR_INPUT  CraneOnMagazin : BOOL; END_VAR {*Irwxp*}
    VAR_INPUT  CraneSucked : BOOL; END_VAR {*Irwxp*}
    VAR_OUTPUT  CraneTurnClockwise : BOOL; END_VAR {*Orwxp*}
    VAR_OUTPUT  CraneTurnCounterclockwise : BOOL; END_VAR {*Orwxp*}
    VAR_INPUT  CraneUp : BOOL; END_VAR {*Irwxp*}
    VAR_OUTPUT  MagazinGreenLamp : BOOL; END_VAR {*Orwxp*}
    VAR_OUTPUT  MagazinSlider : BOOL; END_VAR {*Orwxp*}
    VAR_OUTPUT  MagazinVacuumOff : BOOL; END_VAR {*Orwxp*}
    VAR_OUTPUT  MagazinVacuumOn : BOOL; END_VAR {*Orwxp*}
    VAR_OUTPUT  MagazinWhiteLamp : BOOL; END_VAR {*Orwxp*}
    VAR  SFCInit : BOOL; END_VAR {*Lrwxp*}
    VAR_INPUT  SFCReset : BOOL; END_VAR {*Irwxp*}
    VAR_INPUT  SliderMovedOut : BOOL; END_VAR {*Irwxp*}
    VAR_INPUT  SliderNotMovedOut : BOOL; END_VAR {*Irwxp*}
    VAR_INPUT  StartButtonMagazin : BOOL; END_VAR {*Irwxp*}
    VAR_OUTPUT  StartCommandMagazin : BOOL; END_VAR {*Orwxp*}
    VAR_INPUT  StartVar : BOOL; END_VAR {*Irwxp*}
    VAR_INPUT  WorkpieceReady : BOOL; END_VAR {*Irwxp*}
    VAR  _state : Magazin_states_t; END_VAR {*Lrwxp*}
    VAR  _transit : BOOL; END_VAR {*Lrwxp*}
    VAR  interconnectMagazinStartCommand : BOOL; END_VAR {*Lrwxp*}

    CASE _state OF
        Magazin_states_t#Green_Lamp:
            {* begin(State) *}
            {* begin(onEntry) *}
            _transit := FALSE;
            {* end(onEntry) *}
            {* begin(onActive) *}
            MagazinGreenLamp := TRUE;
            interconnectMagazinStartCommand := FALSE;
            {* end(onActive) *}
            {* begin(transition) *}
            IF TRUE THEN
                _transit := TRUE;
                _state := Magazin_states_t#Magazin_Init;
            END_IF;
            {* end(transition) *}
            {* begin(onExit) *}
            {* end(onExit) *}
            {* end(State) *}

        Magazin_states_t#Init:
            {* begin(State) *}
            {* begin(onEntry) *}
            _transit := FALSE;
            {* end(onEntry) *}
            {* begin(onActive) *}
            {* end(onActive) *}
            {* begin(transition) *}
            IF TRUE THEN
                _transit := TRUE;
                _state := Magazin_states_t#Start_Magazin;
            END_IF;
            {* end(transition) *}
            {* begin(onExit) *}
            {* end(onExit) *}
            {* end(State) *}

        Magazin_states_t#Interstep:
            {* begin(State) *}
            {* begin(onEntry) *}
            _transit := FALSE;
            {* end(onEntry) *}
            {* begin(onActive) *}
            StartCommandMagazin := TRUE;
            {* end(onActive) *}
            {* begin(transition) *}
            IF StartVar THEN
                _transit := TRUE;
                _state := Magazin_states_t#convey;
            END_IF;
            {* end(transition) *}
            {* begin(onExit) *}
            {* end(onExit) *}
            {* end(State) *}

        Magazin_states_t#Magazin_Init:
            {* begin(State) *}
            {* begin(onEntry) *}
            _transit := FALSE;
            {* end(onEntry) *}
            {* begin(onActive) *}
            MagazinSlider := TRUE;
            {* end(onActive) *}
            {* begin(transition) *}
            IF TRUE THEN
                _transit := TRUE;
                _state := Magazin_states_t#Magazin_Init_2;
            END_IF;
            {* end(transition) *}
            {* begin(onExit) *}
            {* end(onExit) *}
            {* end(State) *}

        Magazin_states_t#Magazin_Init_2:
            {* begin(State) *}
            {* begin(onEntry) *}
            _transit := FALSE;
            {* end(onEntry) *}
            {* begin(onActive) *}
            MagazinSlider := FALSE;
            {* end(onActive) *}
            {* begin(transition) *}
            IF TRUE THEN
                _transit := TRUE;
                _state := Magazin_states_t#Interstep;
            END_IF;
            {* end(transition) *}
            {* begin(onExit) *}
            {* end(onExit) *}
            {* end(State) *}

        Magazin_states_t#Slider_Move_Back:
            {* begin(State) *}
            {* begin(onEntry) *}
            _transit := FALSE;
            {* end(onEntry) *}
            {* begin(onActive) *}
            IF ((SliderMovedOut = TRUE) AND (SliderNotMovedOut = FALSE)) THEN
                MagazinSlider := FALSE;
            END_IF;
            {* end(onActive) *}
            {* begin(transition) *}
            IF CraneUp THEN
                _transit := TRUE;
                _state := Magazin_states_t#Step1;
            END_IF;
            {* end(transition) *}
            {* begin(onExit) *}
            {* end(onExit) *}
            {* end(State) *}

        Magazin_states_t#Start_Magazin:
            {* begin(State) *}
            {* begin(onEntry) *}
            _transit := FALSE;
            {* end(onEntry) *}
            {* begin(onActive) *}
            MagazinSlider := FALSE;
            MagazinGreenLamp := FALSE;
            StartVar := FALSE;
            StartCommandMagazin := FALSE;
            IF (StartButtonMagazin = TRUE) THEN
                interconnectMagazinStartCommand := TRUE;
            END_IF;
            {* end(onActive) *}
            {* begin(transition) *}
            IF interconnectMagazinStartCommand THEN
                _transit := TRUE;
                _state := Magazin_states_t#Green_Lamp;
            END_IF;
            {* end(transition) *}
            {* begin(onExit) *}
            {* end(onExit) *}
            {* end(State) *}

        Magazin_states_t#Step0:
            {* begin(State) *}
            {* begin(onEntry) *}
            _transit := FALSE;
            {* end(onEntry) *}
            {* begin(onActive) *}
            {* end(onActive) *}
            {* begin(transition) *}
            IF CraneDown THEN
                _transit := TRUE;
                _state := Magazin_states_t#Slider_Move_Back;
            END_IF;
            {* end(transition) *}
            {* begin(onExit) *}
            {* end(onExit) *}
            {* end(State) *}

        Magazin_states_t#Step1:
            {* begin(State) *}
            {* begin(onEntry) *}
            _transit := FALSE;
            {* end(onEntry) *}
            {* begin(onActive) *}
            {* end(onActive) *}
            {* begin(transition) *}
            IF ((AnalogCranePosition > INT#16160) AND (AnalogCranePosition < INT#16260)) THEN
                _transit := TRUE;
                _state := Magazin_states_t#Interstep;
            END_IF;
            {* end(transition) *}
            {* begin(onExit) *}
            {* end(onExit) *}
            {* end(State) *}

        Magazin_states_t#convey:
            {* begin(State) *}
            {* begin(onEntry) *}
            _transit := FALSE;
            {* end(onEntry) *}
            {* begin(onActive) *}
            IF SliderNotMovedOut THEN
                MagazinSlider := TRUE;
            END_IF;
            {* end(onActive) *}
            {* begin(transition) *}
            IF ((AnalogCranePosition > INT#24290) AND (AnalogCranePosition < INT#24390)) THEN
                _transit := TRUE;
                _state := Magazin_states_t#Step0;
            END_IF;
            {* end(transition) *}
            {* begin(onExit) *}
            {* end(onExit) *}
            {* end(State) *}

            END_CASE;
END_FUNCTION_BLOCK

FUNCTION_BLOCK Conveyor
    VAR  Duration_Conveyor_Runtime : TIME := TIME#4.0s500.0ms; END_VAR {*Lrwxp*}
    VAR  Duration_Conveyor_Test : TIME := TIME#1.0s; END_VAR {*Lrwxp*}
    VAR  SFCInit : BOOL; END_VAR {*Lrwxp*}
    VAR_INPUT  SFCReset : BOOL; END_VAR {*Irwxp*}
    VAR_OUTPUT  SorterConveyorTowardsCrane : BOOL; END_VAR {*Orwxp*}
    VAR_OUTPUT  SorterConveyorTowardsStacker : BOOL; END_VAR {*Orwxp*}
    VAR_OUTPUT  SorterGreenLampConveyor : BOOL; END_VAR {*Orwxp*}
    VAR_INPUT  SorterLightbarrierCraneInterface : BOOL; END_VAR {*Irwxp*}
    VAR_INPUT  SorterStartButton : BOOL; END_VAR {*Irwxp*}
    VAR_INPUT  SorterSwitchManuellAutomatic : BOOL; END_VAR {*Irwxp*}
    VAR_OUTPUT  SorterWhiteLampConveyor : BOOL; END_VAR {*Orwxp*}
    VAR_OUTPUT  StartCommandConveyor : BOOL; END_VAR {*Orwxp*}
    VAR_INPUT  StartVar : BOOL; END_VAR {*Irwxp*}
    VAR  Timer_Conveyor_Runtime : TON; END_VAR {*Lrwxp*}
    VAR  Timer_Conveyor_Test : TON; END_VAR {*Lrwxp*}
    VAR  _state : Conveyor_states_t; END_VAR {*Lrwxp*}
    VAR  _transit : BOOL; END_VAR {*Lrwxp*}
    VAR  interconnectConveyorStartCommand : BOOL; END_VAR {*Lrwxp*}
    VAR  interconnectConveyorTerminationCommand : BOOL; END_VAR {*Lrwxp*}
    VAR  interconnect_Conveyor_Runtime : BOOL; END_VAR {*Lrwxp*}
    VAR  interconnect_Conveyor_Test : BOOL; END_VAR {*Lrwxp*}

    CASE _state OF
        Conveyor_states_t#Conveyor_Init:
            {* begin(State) *}
            {* begin(onEntry) *}
            _transit := FALSE;
            {* end(onEntry) *}
            {* begin(onActive) *}
            SorterConveyorTowardsStacker := TRUE;
            SorterConveyorTowardsCrane := FALSE;
            Timer_Conveyor_Test(IN := TRUE, PT := Duration_Conveyor_Test);
            interconnect_Conveyor_Test := Timer_Conveyor_Test.Q;
            {* end(onActive) *}
            {* begin(transition) *}
            IF interconnect_Conveyor_Test THEN
                _transit := TRUE;
                _state := Conveyor_states_t#Conveyor_init_2;
            END_IF;
            {* end(transition) *}
            {* begin(onExit) *}
            {* end(onExit) *}
            {* end(State) *}

        Conveyor_states_t#Conveyor_Stop_Empty_Magazin:
            {* begin(State) *}
            {* begin(onEntry) *}
            _transit := FALSE;
            {* end(onEntry) *}
            {* begin(onActive) *}
            SorterConveyorTowardsStacker := FALSE;
            SorterConveyorTowardsCrane := FALSE;
            interconnectConveyorStartCommand := FALSE;
            {* end(onActive) *}
            {* begin(transition) *}
            IF TRUE THEN
                _transit := TRUE;
                _state := Conveyor_states_t#Interstep;
            END_IF;
            {* end(transition) *}
            {* begin(onExit) *}
            {* end(onExit) *}
            {* end(State) *}

        Conveyor_states_t#Conveyor_Towards_Stacker:
            {* begin(State) *}
            {* begin(onEntry) *}
            _transit := FALSE;
            {* end(onEntry) *}
            {* begin(onActive) *}
            SorterConveyorTowardsStacker := TRUE;
            SorterConveyorTowardsCrane := FALSE;
            {* end(onActive) *}
            {* begin(transition) *}
            IF TRUE THEN
                _transit := TRUE;
                _state := Conveyor_states_t#Runtime_Conveyor;
            END_IF;
            {* end(transition) *}
            {* begin(onExit) *}
            {* end(onExit) *}
            {* end(State) *}

        Conveyor_states_t#Conveyor_init_2:
            {* begin(State) *}
            {* begin(onEntry) *}
            _transit := FALSE;
            {* end(onEntry) *}
            {* begin(onActive) *}
            SorterConveyorTowardsStacker := FALSE;
            SorterConveyorTowardsCrane := FALSE;
            interconnect_Conveyor_Test := FALSE;
            Timer_Conveyor_Test(IN := FALSE, PT := TIME#);
            {* end(onActive) *}
            {* begin(transition) *}
            IF TRUE THEN
                _transit := TRUE;
                _state := Conveyor_states_t#Interstep;
            END_IF;
            {* end(transition) *}
            {* begin(onExit) *}
            {* end(onExit) *}
            {* end(State) *}

        Conveyor_states_t#Conveyor_pause:
            {* begin(State) *}
            {* begin(onEntry) *}
            _transit := FALSE;
            {* end(onEntry) *}
            {* begin(onActive) *}
            SorterConveyorTowardsStacker := FALSE;
            SorterConveyorTowardsCrane := FALSE;
            interconnect_Conveyor_Runtime := FALSE;
            Timer_Conveyor_Runtime(IN := FALSE, PT := TIME#);
            {* end(onActive) *}
            {* begin(transition) *}
            IF TRUE THEN
                _transit := TRUE;
                _state := Conveyor_states_t#Interstep;
            END_IF;
            {* end(transition) *}
            {* begin(onExit) *}
            {* end(onExit) *}
            {* end(State) *}

        Conveyor_states_t#Green_Lamp:
            {* begin(State) *}
            {* begin(onEntry) *}
            _transit := FALSE;
            {* end(onEntry) *}
            {* begin(onActive) *}
            SorterGreenLampConveyor := TRUE;
            interconnectConveyorStartCommand := FALSE;
            {* end(onActive) *}
            {* begin(transition) *}
            IF TRUE THEN
                _transit := TRUE;
                _state := Conveyor_states_t#Conveyor_Init;
            END_IF;
            {* end(transition) *}
            {* begin(onExit) *}
            {* end(onExit) *}
            {* end(State) *}

        Conveyor_states_t#Init:
            {* begin(State) *}
            {* begin(onEntry) *}
            _transit := FALSE;
            {* end(onEntry) *}
            {* begin(onActive) *}
            {* end(onActive) *}
            {* begin(transition) *}
            IF TRUE THEN
                _transit := TRUE;
                _state := Conveyor_states_t#Start_Conveyor;
            END_IF;
            {* end(transition) *}
            {* begin(onExit) *}
            {* end(onExit) *}
            {* end(State) *}

        Conveyor_states_t#Interstep:
            {* begin(State) *}
            {* begin(onEntry) *}
            _transit := FALSE;
            {* end(onEntry) *}
            {* begin(onActive) *}
            StartCommandConveyor := TRUE;
            {* end(onActive) *}
            {* begin(transition) *}
            IF StartVar THEN
                _transit := TRUE;
                _state := Conveyor_states_t#Step0;
            END_IF;
            {* end(transition) *}
            {* begin(onExit) *}
            {* end(onExit) *}
            {* end(State) *}

        Conveyor_states_t#Runtime_Conveyor:
            {* begin(State) *}
            {* begin(onEntry) *}
            _transit := FALSE;
            {* end(onEntry) *}
            {* begin(onActive) *}
            Timer_Conveyor_Runtime(IN := TRUE, PT := Duration_Conveyor_Runtime);
            interconnect_Conveyor_Runtime := Timer_Conveyor_Runtime.Q;
            {* end(onActive) *}
            {* begin(transition) *}
            IF interconnect_Conveyor_Runtime THEN
                _transit := TRUE;
                _state := Conveyor_states_t#Conveyor_pause;
            END_IF;
            {* end(transition) *}
            {* begin(onExit) *}
            {* end(onExit) *}
            {* end(State) *}

        Conveyor_states_t#Start_Conveyor:
            {* begin(State) *}
            {* begin(onEntry) *}
            _transit := FALSE;
            {* end(onEntry) *}
            {* begin(onActive) *}
            interconnectConveyorTerminationCommand := FALSE;
            SorterConveyorTowardsStacker := FALSE;
            SorterConveyorTowardsCrane := FALSE;
            SorterGreenLampConveyor := FALSE;
            interconnect_Conveyor_Runtime := FALSE;
            interconnect_Conveyor_Test := FALSE;
            Timer_Conveyor_Test(IN := FALSE, PT := TIME#);
            Timer_Conveyor_Runtime(IN := FALSE, PT := TIME#);
            StartVar := FALSE;
            StartCommandConveyor := FALSE;
            IF (SorterStartButton = TRUE) THEN
                interconnectConveyorStartCommand := TRUE;
            END_IF;
            {* end(onActive) *}
            {* begin(transition) *}
            IF interconnectConveyorStartCommand THEN
                _transit := TRUE;
                _state := Conveyor_states_t#Green_Lamp;
            END_IF;
            {* end(transition) *}
            {* begin(onExit) *}
            {* end(onExit) *}
            {* end(State) *}

        Conveyor_states_t#Step0:
            {* begin(State) *}
            {* begin(onEntry) *}
            _transit := FALSE;
            {* end(onEntry) *}
            {* begin(onActive) *}
            {* end(onActive) *}
            {* begin(transition) *}
            IF SorterLightbarrierCraneInterface THEN
                _transit := TRUE;
                _state := Conveyor_states_t#Conveyor_Towards_Stacker;
            ELSEIF NOT SorterLightbarrierCraneInterface THEN
                _transit := TRUE;
                _state := Conveyor_states_t#Conveyor_Stop_Empty_Magazin;
            END_IF;
            {* end(transition) *}
            {* begin(onExit) *}
            {* end(onExit) *}
            {* end(State) *}

            END_CASE;
END_FUNCTION_BLOCK

PROGRAM Main

VAR  Actuator_AnalogCranePressure : INT; END_VAR {*Lrwxp*}
VAR  Actuator_CraneLower : BOOL; END_VAR {*Lrwxp*}
VAR  Actuator_CraneTurnClockwise : BOOL; END_VAR {*Lrwxp*}
VAR  Actuator_CraneTurnCounterclockwise : BOOL; END_VAR {*Lrwxp*}
VAR  Actuator_MagazinGreenLamp : BOOL; END_VAR {*Lrwxp*}
VAR  Actuator_MagazinSlider : BOOL; END_VAR {*Lrwxp*}
VAR  Actuator_MagazinVacuumOff : BOOL; END_VAR {*Lrwxp*}
VAR  Actuator_MagazinVacuumOn : BOOL; END_VAR {*Lrwxp*}
VAR  Actuator_MagazinWhiteLamp : BOOL; END_VAR {*Lrwxp*}
VAR  Actuator_PusherY1 : BOOL; END_VAR {*Lrwxp*}
VAR  Actuator_PusherY2 : BOOL; END_VAR {*Lrwxp*}
VAR  Actuator_SorterConveyorTowardsCrane : BOOL; END_VAR {*Lrwxp*}
VAR  Actuator_SorterConveyorTowardsStacker : BOOL; END_VAR {*Lrwxp*}
VAR  Actuator_SorterGreenLampConveyor : BOOL; END_VAR {*Lrwxp*}
VAR  Actuator_SorterWhiteLampConveyor : BOOL; END_VAR {*Lrwxp*}
VAR  Actuator_StampGreenLamp : BOOL; END_VAR {*Lrwxp*}
VAR  Actuator_StampPusher : BOOL; END_VAR {*Lrwxp*}
VAR  Actuator_StampSliderMovedIn : BOOL; END_VAR {*Lrwxp*}
VAR  Actuator_StampSliderMovedOut : BOOL; END_VAR {*Lrwxp*}
VAR  Actuator_StampWhiteLamp : BOOL; END_VAR {*Lrwxp*}
VAR  Conveyor : Conveyor; END_VAR {*Lrwxp*}
VAR  Crane : Crane; END_VAR {*Lrwxp*}
VAR  Mag : Magazin; END_VAR {*Lrwxp*}
VAR  Pusher : Pusher; END_VAR {*Lrwxp*}
VAR  Sensor_AnalogCranePosition : INT; END_VAR {*Lrwxp*}
VAR  Sensor_CraneDown : BOOL; END_VAR {*Lrwxp*}
VAR  Sensor_CraneOnConveyor : BOOL; END_VAR {*Lrwxp*}
VAR  Sensor_CraneOnMagazin : BOOL; END_VAR {*Lrwxp*}
VAR  Sensor_CranePosition : BOOL; END_VAR {*Lrwxp*}
VAR  Sensor_CranePositionStamp : BOOL; END_VAR {*Lrwxp*}
VAR  Sensor_CraneSucked : BOOL; END_VAR {*Lrwxp*}
VAR  Sensor_CraneUp : BOOL; END_VAR {*Lrwxp*}
VAR  Sensor_MagazinCapacitiveSensor : BOOL; END_VAR {*Lrwxp*}
VAR  Sensor_MagazinEmergencyStop : BOOL; END_VAR {*Lrwxp*}
VAR  Sensor_MagazinOpticalSensor : BOOL; END_VAR {*Lrwxp*}
VAR  Sensor_MagazinSwitchManuellAutomatic : BOOL; END_VAR {*Lrwxp*}
VAR  Sensor_SliderMovedOut : BOOL; END_VAR {*Lrwxp*}
VAR  Sensor_SliderNotMovedOut : BOOL; END_VAR {*Lrwxp*}
VAR  Sensor_SorterCapacitiveSensorPusher1 : BOOL; END_VAR {*Lrwxp*}
VAR  Sensor_SorterCapacitiveSensorPusher2 : BOOL; END_VAR {*Lrwxp*}
VAR  Sensor_SorterEmergencyStop : BOOL; END_VAR {*Lrwxp*}
VAR  Sensor_SorterLightbarrierCraneInterface : BOOL; END_VAR {*Lrwxp*}
VAR  Sensor_SorterLightnessSensorPusher1 : BOOL; END_VAR {*Lrwxp*}
VAR  Sensor_SorterLightnessSensorPusher2 : BOOL; END_VAR {*Lrwxp*}
VAR  Sensor_SorterLightnessSensorPusher3 : BOOL; END_VAR {*Lrwxp*}
VAR  Sensor_SorterLightnesssensorCraneInterfaceInverse : BOOL; END_VAR {*Lrwxp*}
VAR  Sensor_SorterPusher1MovedIn : BOOL; END_VAR {*Lrwxp*}
VAR  Sensor_SorterPusher1MovedOut : BOOL; END_VAR {*Lrwxp*}
VAR  Sensor_SorterPusher2MovedIn : BOOL; END_VAR {*Lrwxp*}
VAR  Sensor_SorterPusher2MovedOut : BOOL; END_VAR {*Lrwxp*}
VAR  Sensor_SorterStartButton : BOOL; END_VAR {*Lrwxp*}
VAR  Sensor_SorterSwitchManuellAutomatic : BOOL; END_VAR {*Lrwxp*}
VAR  Sensor_StampEmergencyStop : BOOL; END_VAR {*Lrwxp*}
VAR  Sensor_StampLowered : BOOL; END_VAR {*Lrwxp*}
VAR  Sensor_StampSliderFilled : BOOL; END_VAR {*Lrwxp*}
VAR  Sensor_StampSliderSensorMovedIn : BOOL; END_VAR {*Lrwxp*}
VAR  Sensor_StampSliderSensorMovedOut : BOOL; END_VAR {*Lrwxp*}
VAR  Sensor_StampStartButton : BOOL; END_VAR {*Lrwxp*}
VAR  Sensor_StampSwitchManuellAutomatic : BOOL; END_VAR {*Lrwxp*}
VAR  Sensor_StampUp : BOOL; END_VAR {*Lrwxp*}
VAR  Sensor_StartButtonMagazin : BOOL; END_VAR {*Lrwxp*}
VAR  Sensor_WorkpieceReady : BOOL; END_VAR {*Lrwxp*}
VAR  Stamp : Stamp; END_VAR {*Lrwxp*}
Mag.SliderNotMovedOut := Sensor_SliderNotMovedOut;
Mag.SliderMovedOut := Sensor_SliderMovedOut;
Mag.CraneOnMagazin := Sensor_CraneOnMagazin;
Mag.CraneDown := Sensor_CraneDown;
Mag.CraneUp := Sensor_CraneUp;
Mag.CraneOnConveyor := Sensor_CraneOnConveyor;
Mag.WorkpieceReady := Sensor_WorkpieceReady;
Mag.AnalogCranePosition := Sensor_AnalogCranePosition;
Mag.StartButtonMagazin := Sensor_StartButtonMagazin;
Actuator_MagazinSlider := Mag.MagazinSlider;
Actuator_MagazinGreenLamp := Mag.MagazinGreenLamp;
Crane.CraneUp := Sensor_CraneUp;
Crane.CraneDown := Sensor_CraneDown;
Crane.CraneSucked := Sensor_CraneSucked;
Crane.MagazinCapacitiveSensor := Sensor_MagazinCapacitiveSensor;
Crane.SliderMovedOut := Sensor_SliderMovedOut;
Crane.WorkpieceReady := Sensor_WorkpieceReady;
Crane.MagazinOpticalSensor := Sensor_MagazinOpticalSensor;
Crane.StampSliderFilled := Sensor_StampSliderFilled;
Crane.StampSliderSensorMovedOut := Sensor_StampSliderSensorMovedOut;
Crane.StampLowered := Sensor_StampLowered;
Crane.AnalogCranePosition := Sensor_AnalogCranePosition;
Crane.StartButtonMagazin := Sensor_StartButtonMagazin;
Actuator_CraneTurnCounterclockwise := Crane.CraneTurnCounterclockwise;
Actuator_CraneTurnClockwise := Crane.CraneTurnClockwise;
Actuator_CraneLower := Crane.CraneLower;
Actuator_MagazinVacuumOff := Crane.MagazinVacuumOff;
Actuator_MagazinVacuumOn := Crane.MagazinVacuumOn;
Actuator_AnalogCranePressure := Crane.AnalogCranePressure;
Stamp.StampSliderSensorMovedOut := Sensor_StampSliderSensorMovedOut;
Stamp.StampSliderSensorMovedIn := Sensor_StampSliderSensorMovedIn;
Stamp.StampSliderFilled := Sensor_StampSliderFilled;
Stamp.StampUp := Sensor_StampUp;
Stamp.StampLowered := Sensor_StampLowered;
Stamp.CraneDown := Sensor_CraneDown;
Stamp.CraneUp := Sensor_CraneUp;
Stamp.CraneSucked := Sensor_CraneSucked;
Stamp.CranePositionStamp := Sensor_CranePositionStamp;
Stamp.CraneOnConveyor := Sensor_CraneOnConveyor;
Stamp.AnalogCranePosition := Sensor_AnalogCranePosition;
Stamp.StampStartButton := Sensor_StampStartButton;
Actuator_StampSliderMovedOut := Stamp.StampSliderMovedOut;
Actuator_StampSliderMovedIn := Stamp.StampSliderMovedIn;
Actuator_StampWhiteLamp := Stamp.StampWhiteLamp;
Actuator_StampPusher := Stamp.StampPusher;
Actuator_StampGreenLamp := Stamp.StampGreenLamp;
Conveyor.SorterStartButton := Sensor_SorterStartButton;
Conveyor.SorterSwitchManuellAutomatic := Sensor_SorterSwitchManuellAutomatic;
Conveyor.SorterLightbarrierCraneInterface := Sensor_SorterLightbarrierCraneInterface;
Actuator_SorterConveyorTowardsStacker := Conveyor.SorterConveyorTowardsStacker;
Actuator_SorterConveyorTowardsCrane := Conveyor.SorterConveyorTowardsCrane;
Actuator_SorterGreenLampConveyor := Conveyor.SorterGreenLampConveyor;
Actuator_SorterWhiteLampConveyor := Conveyor.SorterWhiteLampConveyor;
Pusher.SorterLightnesssensorCraneInterfaceInverse := Sensor_SorterLightnesssensorCraneInterfaceInverse;
Pusher.SorterLightbarrierCraneInterface := Sensor_SorterLightbarrierCraneInterface;
Pusher.SorterCapacitiveSensorPusher1 := Sensor_SorterCapacitiveSensorPusher1;
Pusher.SorterLightnessSensorPusher1 := Sensor_SorterLightnessSensorPusher1;
Pusher.SorterCapacitiveSensorPusher2 := Sensor_SorterCapacitiveSensorPusher2;
Pusher.SorterLightnessSensorPusher2 := Sensor_SorterLightnessSensorPusher2;
Pusher.SorterLightnessSensorPusher3 := Sensor_SorterLightnessSensorPusher3;
Pusher.SorterPusher1MovedOut := Sensor_SorterPusher1MovedOut;
Pusher.SorterPusher1MovedIn := Sensor_SorterPusher1MovedIn;
Pusher.SorterPusher2MovedOut := Sensor_SorterPusher2MovedOut;
Pusher.SorterPusher2MovedIn := Sensor_SorterPusher2MovedIn;
Pusher.SorterStartButton := Sensor_SorterStartButton;
Actuator_PusherY1 := Pusher.PusherY1;
Actuator_PusherY2 := Pusher.PusherY2;
IF ((Sensor_SorterEmergencyStop AND Sensor_StampEmergencyStop) AND Sensor_MagazinEmergencyStop) THEN
    Mag();
    Crane();
    Stamp();
    Conveyor();
    Pusher();
    IF ((Actuator_SorterGreenLampConveyor AND Actuator_MagazinGreenLamp) AND Actuator_StampGreenLamp) THEN
        IF (((Stamp.StartCommandStamp AND Crane.StartCommandCrane) AND Conveyor.StartCommandConveyor) AND Mag.StartCommandMagazin) THEN
            Crane.StartVar := TRUE;
            Conveyor.StartVar := TRUE;
            Mag.StartVar := TRUE;
            Pusher.StartVar := TRUE;
            Stamp.StartVar := TRUE;
        END_IF;
    END_IF;
    Crane.SFCReset := FALSE;
    Conveyor.SFCReset := FALSE;
    Mag.SFCReset := FALSE;
    Pusher.SFCReset := FALSE;
    Stamp.SFCReset := FALSE;
ELSEIF ((NOT Sensor_SorterEmergencyStop OR NOT Sensor_StampEmergencyStop) OR NOT Sensor_MagazinEmergencyStop) THEN
    Actuator_MagazinSlider := FALSE;
    Actuator_CraneLower := FALSE;
    Actuator_MagazinVacuumOn := FALSE;
    Actuator_MagazinVacuumOff := TRUE;
    Actuator_MagazinGreenLamp := FALSE;
    Actuator_CraneTurnCounterclockwise := FALSE;
    Actuator_CraneTurnClockwise := FALSE;
    Actuator_SorterConveyorTowardsStacker := FALSE;
    Actuator_SorterConveyorTowardsCrane := FALSE;
    Actuator_SorterGreenLampConveyor := FALSE;
    Actuator_PusherY1 := FALSE;
    Actuator_PusherY2 := FALSE;
    Actuator_StampSliderMovedOut := TRUE;
    Actuator_StampSliderMovedIn := FALSE;
    Actuator_StampGreenLamp := FALSE;
    Actuator_StampPusher := FALSE;
    Actuator_AnalogCranePressure := INT#0;
    Crane.SFCReset := TRUE;
    Conveyor.SFCReset := TRUE;
    Mag.SFCReset := TRUE;
    Pusher.SFCReset := TRUE;
    Stamp.SFCReset := TRUE;
    Crane.StartVar := FALSE;
    Conveyor.StartVar := FALSE;
    Mag.StartVar := FALSE;
    Pusher.StartVar := FALSE;
    Stamp.StartVar := FALSE;
END_IF;
END_PROGRAM
FUNCTION_BLOCK Stamp
VAR_INPUT  AnalogCranePosition : INT; END_VAR {*Irwxp*}
VAR_INPUT  CraneDown : BOOL; END_VAR {*Irwxp*}
VAR_INPUT  CraneOnConveyor : BOOL; END_VAR {*Irwxp*}
VAR_INPUT  CranePositionStamp : BOOL; END_VAR {*Irwxp*}
VAR_INPUT  CraneSucked : BOOL; END_VAR {*Irwxp*}
VAR_INPUT  CraneUp : BOOL; END_VAR {*Irwxp*}
VAR  Duration : TIME := TIME#500.0ms; END_VAR {*Lrwxp*}
VAR  SFCInit : BOOL; END_VAR {*Lrwxp*}
VAR_INPUT  SFCReset : BOOL; END_VAR {*Irwxp*}
VAR_OUTPUT  StampGreenLamp : BOOL; END_VAR {*Orwxp*}
VAR_INPUT  StampLowered : BOOL; END_VAR {*Irwxp*}
VAR_OUTPUT  StampPressure : BOOL; END_VAR {*Orwxp*}
VAR_OUTPUT  StampPusher : BOOL; END_VAR {*Orwxp*}
VAR_INPUT  StampSliderFilled : BOOL; END_VAR {*Irwxp*}
VAR_OUTPUT  StampSliderMovedIn : BOOL; END_VAR {*Orwxp*}
VAR_OUTPUT  StampSliderMovedOut : BOOL; END_VAR {*Orwxp*}
VAR_INPUT  StampSliderSensorMovedIn : BOOL; END_VAR {*Irwxp*}
VAR_INPUT  StampSliderSensorMovedOut : BOOL; END_VAR {*Irwxp*}
VAR_INPUT  StampStartButton : BOOL; END_VAR {*Irwxp*}
VAR_INPUT  StampUp : BOOL; END_VAR {*Irwxp*}
VAR_OUTPUT  StampWhiteLamp : BOOL; END_VAR {*Orwxp*}
VAR_OUTPUT  StartCommandStamp : BOOL; END_VAR {*Orwxp*}
VAR_INPUT  StartVar : BOOL; END_VAR {*Irwxp*}
VAR  Timer : TON; END_VAR {*Lrwxp*}
VAR  _state : Stamp_states_t; END_VAR {*Lrwxp*}
VAR  _transit : BOOL; END_VAR {*Lrwxp*}
VAR  interconnect : BOOL; END_VAR {*Lrwxp*}
VAR  interconnectStampStartCommand : BOOL; END_VAR {*Lrwxp*}

CASE _state OF
    Stamp_states_t#Green_Lamp:
        {* begin(State) *}
        {* begin(onEntry) *}
        _transit := FALSE;
        {* end(onEntry) *}
        {* begin(onActive) *}
        StampGreenLamp := TRUE;
        interconnectStampStartCommand := FALSE;
        {* end(onActive) *}
        {* begin(transition) *}
        IF TRUE THEN
            _transit := TRUE;
            _state := Stamp_states_t#Stamp_Init_1;
        END_IF;
        {* end(transition) *}
        {* begin(onExit) *}
        {* end(onExit) *}
        {* end(State) *}

    Stamp_states_t#Init:
        {* begin(State) *}
        {* begin(onEntry) *}
        _transit := FALSE;
        {* end(onEntry) *}
        {* begin(onActive) *}
        {* end(onActive) *}
        {* begin(transition) *}
        IF TRUE THEN
            _transit := TRUE;
            _state := Stamp_states_t#Start_Stamp;
        END_IF;
        {* end(transition) *}
        {* begin(onExit) *}
        {* end(onExit) *}
        {* end(State) *}

    Stamp_states_t#Interstep:
        {* begin(State) *}
        {* begin(onEntry) *}
        _transit := FALSE;
        {* end(onEntry) *}
        {* begin(onActive) *}
        StartCommandStamp := TRUE;
        {* end(onActive) *}
        {* begin(transition) *}
        IF StartVar THEN
            _transit := TRUE;
            _state := Stamp_states_t#Intertsep_2;
        END_IF;
        {* end(transition) *}
        {* begin(onExit) *}
        {* end(onExit) *}
        {* end(State) *}

    Stamp_states_t#Intertsep_2:
        {* begin(State) *}
        {* begin(onEntry) *}
        _transit := FALSE;
        {* end(onEntry) *}
        {* begin(onActive) *}
        {* end(onActive) *}
        {* begin(transition) *}
        IF StampSliderFilled THEN
            _transit := TRUE;
            _state := Stamp_states_t#Step0;
        END_IF;
        {* end(transition) *}
        {* begin(onExit) *}
        {* end(onExit) *}
        {* end(State) *}

    Stamp_states_t#StampProcess:
        {* begin(State) *}
        {* begin(onEntry) *}
        _transit := FALSE;
        {* end(onEntry) *}
        {* begin(onActive) *}
        StampSliderMovedIn := FALSE;
        StampPusher := TRUE;
        {* end(onActive) *}
        {* begin(transition) *}
        IF StampLowered THEN
            _transit := TRUE;
            _state := Stamp_states_t#Step1;
        END_IF;
        {* end(transition) *}
        {* begin(onExit) *}
        {* end(onExit) *}
        {* end(State) *}

    Stamp_states_t#StampSliderBack:
        {* begin(State) *}
        {* begin(onEntry) *}
        _transit := FALSE;
        {* end(onEntry) *}
        {* begin(onActive) *}
        StampSliderMovedIn := TRUE;
        StampSliderMovedOut := FALSE;
        {* end(onActive) *}
        {* begin(transition) *}
        IF StampSliderSensorMovedIn THEN
            _transit := TRUE;
            _state := Stamp_states_t#StampProcess;
        END_IF;
        {* end(transition) *}
        {* begin(onExit) *}
        {* end(onExit) *}
        {* end(State) *}

    Stamp_states_t#StampSliderForward:
        {* begin(State) *}
        {* begin(onEntry) *}
        _transit := FALSE;
        {* end(onEntry) *}
        {* begin(onActive) *}
        StampPusher := FALSE;
        StampSliderMovedOut := TRUE;
        IF ((StampLowered = FALSE) AND (StampUp = TRUE)) THEN
            interconnect := FALSE;
        END_IF;
        Timer(IN := FALSE, PT := TIME#1.0ms);
        {* end(onActive) *}
        {* begin(transition) *}
        IF StampSliderMovedOut THEN
            _transit := TRUE;
            _state := Stamp_states_t#Step2;
        END_IF;
        {* end(transition) *}
        {* begin(onExit) *}
        {* end(onExit) *}
        {* end(State) *}

    Stamp_states_t#Stamp_Init_1:
        {* begin(State) *}
        {* begin(onEntry) *}
        _transit := FALSE;
        {* end(onEntry) *}
        {* begin(onActive) *}
        StampSliderMovedIn := TRUE;
        StampSliderMovedOut := FALSE;
        {* end(onActive) *}
        {* begin(transition) *}
        IF StampSliderSensorMovedIn THEN
            _transit := TRUE;
            _state := Stamp_states_t#Stamp_Init_2;
        END_IF;
        {* end(transition) *}
        {* begin(onExit) *}
        {* end(onExit) *}
        {* end(State) *}

    Stamp_states_t#Stamp_Init_2:
        {* begin(State) *}
        {* begin(onEntry) *}
        _transit := FALSE;
        {* end(onEntry) *}
        {* begin(onActive) *}
        StampSliderMovedIn := FALSE;
        StampSliderMovedOut := TRUE;
        {* end(onActive) *}
        {* begin(transition) *}
        IF StampSliderSensorMovedOut THEN
            _transit := TRUE;
            _state := Stamp_states_t#Stamp_Init_3;
        END_IF;
        {* end(transition) *}
        {* begin(onExit) *}
        {* end(onExit) *}
        {* end(State) *}

    Stamp_states_t#Stamp_Init_3:
        {* begin(State) *}
        {* begin(onEntry) *}
        _transit := FALSE;
        {* end(onEntry) *}
        {* begin(onActive) *}
        StampPusher := TRUE;
        {* end(onActive) *}
        {* begin(transition) *}
        IF StampLowered THEN
            _transit := TRUE;
            _state := Stamp_states_t#Stamp_Init_4;
        END_IF;
        {* end(transition) *}
        {* begin(onExit) *}
        {* end(onExit) *}
        {* end(State) *}

    Stamp_states_t#Stamp_Init_4:
        {* begin(State) *}
        {* begin(onEntry) *}
        _transit := FALSE;
        {* end(onEntry) *}
        {* begin(onActive) *}
        StampPusher := FALSE;
        {* end(onActive) *}
        {* begin(transition) *}
        IF StampUp THEN
            _transit := TRUE;
            _state := Stamp_states_t#Interstep;
        END_IF;
        {* end(transition) *}
        {* begin(onExit) *}
        {* end(onExit) *}
        {* end(State) *}

    Stamp_states_t#Start_Stamp:
        {* begin(State) *}
        {* begin(onEntry) *}
        _transit := FALSE;
        {* end(onEntry) *}
        {* begin(onActive) *}
        StampSliderMovedOut := FALSE;
        StampSliderMovedIn := FALSE;
        StampPusher := FALSE;
        StampGreenLamp := FALSE;
        StampPressure := FALSE;
        StartCommandStamp := FALSE;
        IF (StampStartButton = TRUE) THEN
            interconnectStampStartCommand := TRUE;
        END_IF;
        {* end(onActive) *}
        {* begin(transition) *}
        IF interconnectStampStartCommand THEN
            _transit := TRUE;
            _state := Stamp_states_t#Green_Lamp;
        END_IF;
        {* end(transition) *}
        {* begin(onExit) *}
        {* end(onExit) *}
        {* end(State) *}

    Stamp_states_t#Step0:
        {* begin(State) *}
        {* begin(onEntry) *}
        _transit := FALSE;
        {* end(onEntry) *}
        {* begin(onActive) *}
        {* end(onActive) *}
        {* begin(transition) *}
        IF CraneUp THEN
            _transit := TRUE;
            _state := Stamp_states_t#StampSliderBack;
        END_IF;
        {* end(transition) *}
        {* begin(onExit) *}
        {* end(onExit) *}
        {* end(State) *}

    Stamp_states_t#Step1:
        {* begin(State) *}
        {* begin(onEntry) *}
        _transit := FALSE;
        {* end(onEntry) *}
        {* begin(onActive) *}
        Timer(IN := StampLowered, PT := TIME#);
        interconnect := Timer.Q;
        {* end(onActive) *}
        {* begin(transition) *}
        IF interconnect THEN
            _transit := TRUE;
            _state := Stamp_states_t#StampSliderForward;
        END_IF;
        {* end(transition) *}
        {* begin(onExit) *}
        {* end(onExit) *}
        {* end(State) *}

    Stamp_states_t#Step2:
        {* begin(State) *}
        {* begin(onEntry) *}
        _transit := FALSE;
        {* end(onEntry) *}
        {* begin(onActive) *}
        {* end(onActive) *}
        {* begin(transition) *}
        IF (((AnalogCranePosition > INT#16160) AND (AnalogCranePosition < INT#16260)) AND NOT StampSliderFilled) THEN
            _transit := TRUE;
            _state := Stamp_states_t#Interstep;
        END_IF;
        {* end(transition) *}
        {* begin(onExit) *}
        {* end(onExit) *}
        {* end(State) *}

    END_CASE;
END_FUNCTION_BLOCK

FUNCTION_BLOCK Pusher
VAR  Duration2 : TIME := TIME#2.0s; END_VAR {*Lrwxp*}
VAR  Duration3 : TIME := TIME#200.0ms; END_VAR {*Lrwxp*}
VAR  Duration_Slide1_Black : TIME := TIME#950.0ms; END_VAR {*Lrwxp*}
VAR  Duration_Slide1_Metal : TIME := TIME#300.0ms; END_VAR {*Lrwxp*}
VAR  Duration_Slide1_White : TIME := TIME#300.0ms; END_VAR {*Lrwxp*}
VAR  Duration_Slide2_Black : TIME := TIME#2.0s; END_VAR {*Lrwxp*}
VAR  Duration_Slide2_Metal : TIME := TIME#370.0ms; END_VAR {*Lrwxp*}
VAR  Duration_Slide2_White : TIME := TIME#370.0ms; END_VAR {*Lrwxp*}
VAR  Priority_Var_Black : INT := INT#3; END_VAR {*Lrwxp*}
VAR  Priority_Var_Metal : INT := INT#3; END_VAR {*Lrwxp*}
VAR  Priority_Var_White : INT := INT#3; END_VAR {*Lrwxp*}
VAR_OUTPUT  PusherY1 : BOOL; END_VAR {*Orwxp*}
VAR_OUTPUT  PusherY2 : BOOL; END_VAR {*Orwxp*}
VAR  SFCInit : BOOL; END_VAR {*Lrwxp*}
VAR_INPUT  SFCReset : BOOL; END_VAR {*Irwxp*}
VAR  Slide1_black : INT := INT#1; END_VAR {*Lrwxp*}
VAR  Slide1_metal : INT := INT#1; END_VAR {*Lrwxp*}
VAR  Slide1_white : INT := INT#1; END_VAR {*Lrwxp*}
VAR  Slide2_black : INT := INT#1; END_VAR {*Lrwxp*}
VAR  Slide2_metal : INT := INT#1; END_VAR {*Lrwxp*}
VAR  Slide2_white : INT := INT#1; END_VAR {*Lrwxp*}
VAR  Slide3_black : INT := INT#1; END_VAR {*Lrwxp*}
VAR  Slide3_metal : INT := INT#1; END_VAR {*Lrwxp*}
VAR  Slide3_white : INT := INT#1; END_VAR {*Lrwxp*}
VAR_INPUT  SorterCapacitiveSensorPusher1 : BOOL; END_VAR {*Irwxp*}
VAR_INPUT  SorterCapacitiveSensorPusher2 : BOOL; END_VAR {*Irwxp*}
VAR_INPUT  SorterLightbarrierCraneInterface : BOOL; END_VAR {*Irwxp*}
VAR_INPUT  SorterLightnessSensorPusher1 : BOOL; END_VAR {*Irwxp*}
VAR_INPUT  SorterLightnessSensorPusher2 : BOOL; END_VAR {*Irwxp*}
VAR_INPUT  SorterLightnessSensorPusher3 : BOOL; END_VAR {*Irwxp*}
VAR_INPUT  SorterLightnesssensorCraneInterfaceInverse : BOOL; END_VAR {*Irwxp*}
VAR_INPUT  SorterPusher1MovedIn : BOOL; END_VAR {*Irwxp*}
VAR_INPUT  SorterPusher1MovedOut : BOOL; END_VAR {*Irwxp*}
VAR_INPUT  SorterPusher2MovedIn : BOOL; END_VAR {*Irwxp*}
VAR_INPUT  SorterPusher2MovedOut : BOOL; END_VAR {*Irwxp*}
VAR_INPUT  SorterStartButton : BOOL; END_VAR {*Irwxp*}
VAR_INPUT  StartVar : BOOL; END_VAR {*Irwxp*}
VAR  Timer2 : TON; END_VAR {*Lrwxp*}
VAR  Timer3 : TON; END_VAR {*Lrwxp*}
VAR  Timer_Slide1_Black : TON; END_VAR {*Lrwxp*}
VAR  Timer_Slide1_Metal : TON; END_VAR {*Lrwxp*}
VAR  Timer_Slide1_White : TON; END_VAR {*Lrwxp*}
VAR  Timer_Slide2_Black : TON; END_VAR {*Lrwxp*}
VAR  Timer_Slide2_Metal : TON; END_VAR {*Lrwxp*}
VAR  Timer_Slide2_White : TON; END_VAR {*Lrwxp*}
VAR  _state : Pusher_states_t; END_VAR {*Lrwxp*}
VAR  _transit : BOOL; END_VAR {*Lrwxp*}
VAR  interconnect2 : BOOL; END_VAR {*Lrwxp*}
VAR  interconnect3 : BOOL; END_VAR {*Lrwxp*}
VAR  interconnect_Slide1_Black : BOOL; END_VAR {*Lrwxp*}
VAR  interconnect_Slide1_Metal : BOOL; END_VAR {*Lrwxp*}
VAR  interconnect_Slide1_White : BOOL; END_VAR {*Lrwxp*}
VAR  interconnect_Slide2_Black : BOOL; END_VAR {*Lrwxp*}
VAR  interconnect_Slide2_Metal : BOOL; END_VAR {*Lrwxp*}
VAR  interconnect_Slide2_White : BOOL; END_VAR {*Lrwxp*}

CASE _state OF
    Pusher_states_t#Check_For_Black:
        {* begin(State) *}
        {* begin(onEntry) *}
        _transit := FALSE;
        {* end(onEntry) *}
        {* begin(onActive) *}
        {* end(onActive) *}
        {* begin(transition) *}
        IF ((Slide2_black = INT#1) AND (Priority_Var_Black = INT#2)) THEN
            _transit := TRUE;
            _state := Pusher_states_t#Second_Slide_black_workpieces;
        ELSEIF ((Slide3_black = INT#1) AND (Priority_Var_Black = INT#3)) THEN
            _transit := TRUE;
            _state := Pusher_states_t#Third_Slide_black_workpieces;
        ELSEIF ((Slide1_black = INT#1) AND (Priority_Var_Black = INT#1)) THEN
            _transit := TRUE;
            _state := Pusher_states_t#First_Slide_black_workpieces;
        END_IF;
        {* end(transition) *}
        {* begin(onExit) *}
        {* end(onExit) *}
        {* end(State) *}

    Pusher_states_t#Check_For_Metal:
        {* begin(State) *}
        {* begin(onEntry) *}
        _transit := FALSE;
        {* end(onEntry) *}
        {* begin(onActive) *}
        {* end(onActive) *}
        {* begin(transition) *}
        IF ((Slide3_metal = INT#1) AND (Priority_Var_Metal = INT#3)) THEN
            _transit := TRUE;
            _state := Pusher_states_t#Third_Slide_metal_workpieces;
        ELSEIF ((Slide2_metal = INT#1) AND (Priority_Var_Metal = INT#2)) THEN
            _transit := TRUE;
            _state := Pusher_states_t#Second_Slide_metal_workpieces;
        ELSEIF ((Slide1_metal = INT#1) AND (Priority_Var_Metal = INT#1)) THEN
            _transit := TRUE;
            _state := Pusher_states_t#First_Slide_metal_workpieces;
        END_IF;
        {* end(transition) *}
        {* begin(onExit) *}
        {* end(onExit) *}
        {* end(State) *}

    Pusher_states_t#Check_For_White:
        {* begin(State) *}
        {* begin(onEntry) *}
        _transit := FALSE;
        {* end(onEntry) *}
        {* begin(onActive) *}
        {* end(onActive) *}
        {* begin(transition) *}
        IF ((Slide1_white = INT#1) AND (Priority_Var_White = INT#1)) THEN
            _transit := TRUE;
            _state := Pusher_states_t#First_Slide_white_workpieces;
        ELSEIF ((Slide3_white = INT#1) AND (Priority_Var_White = INT#3)) THEN
            _transit := TRUE;
            _state := Pusher_states_t#Third_Slide_white_workpieces;
        ELSEIF ((Slide2_white = INT#1) AND (Priority_Var_White = INT#2)) THEN
            _transit := TRUE;
            _state := Pusher_states_t#Second_Slide_white_workpieces;
        END_IF;
        {* end(transition) *}
        {* begin(onExit) *}
        {* end(onExit) *}
        {* end(State) *}

    Pusher_states_t#First_Slide_Timer_Black:
        {* begin(State) *}
        {* begin(onEntry) *}
        _transit := FALSE;
        {* end(onEntry) *}
        {* begin(onActive) *}
        IF (SorterLightnesssensorCraneInterfaceInverse = TRUE) THEN
            Timer_Slide1_Black(IN := SorterLightnesssensorCraneInterfaceInverse, PT := Duration_Slide1_Black);
            interconnect_Slide1_Black := Timer_Slide1_Black.Q;
        END_IF;
        {* end(onActive) *}
        {* begin(transition) *}
        IF interconnect_Slide1_Black THEN
            _transit := TRUE;
            _state := Pusher_states_t#PusherY1_Move_Out_Black;
        END_IF;
        {* end(transition) *}
        {* begin(onExit) *}
        {* end(onExit) *}
        {* end(State) *}

    Pusher_states_t#First_Slide_Timer_Metal:
        {* begin(State) *}
        {* begin(onEntry) *}
        _transit := FALSE;
        {* end(onEntry) *}
        {* begin(onActive) *}
        Timer_Slide1_Metal(IN := TRUE, PT := Duration_Slide1_Metal);
        interconnect_Slide1_Metal := Timer_Slide1_Metal.Q;
        {* end(onActive) *}
        {* begin(transition) *}
        IF interconnect_Slide1_Metal THEN
            _transit := TRUE;
            _state := Pusher_states_t#PusherY1_Move_Out_Metal;
        END_IF;
        {* end(transition) *}
        {* begin(onExit) *}
        {* end(onExit) *}
        {* end(State) *}

    Pusher_states_t#First_Slide_Timer_White:
        {* begin(State) *}
        {* begin(onEntry) *}
        _transit := FALSE;
        {* end(onEntry) *}
        {* begin(onActive) *}
        Timer_Slide1_White(IN := TRUE, PT := Duration_Slide1_White);
        interconnect_Slide1_White := Timer_Slide1_White.Q;
        {* end(onActive) *}
        {* begin(transition) *}
        IF interconnect_Slide1_White THEN
            _transit := TRUE;
            _state := Pusher_states_t#PusherY1_Move_Out_White;
        END_IF;
        {* end(transition) *}
        {* begin(onExit) *}
        {* end(onExit) *}
        {* end(State) *}

    Pusher_states_t#First_Slide_black_workpieces:
        {* begin(State) *}
        {* begin(onEntry) *}
        _transit := FALSE;
        {* end(onEntry) *}
        {* begin(onActive) *}
        {* end(onActive) *}
        {* begin(transition) *}
        IF TRUE THEN
            _transit := TRUE;
            _state := Pusher_states_t#First_Slide_Timer_Black;
        END_IF;
        {* end(transition) *}
        {* begin(onExit) *}
        {* end(onExit) *}
        {* end(State) *}

    Pusher_states_t#First_Slide_metal_workpieces:
        {* begin(State) *}
        {* begin(onEntry) *}
        _transit := FALSE;
        {* end(onEntry) *}
        {* begin(onActive) *}
        {* end(onActive) *}
        {* begin(transition) *}
        IF TRUE THEN
            _transit := TRUE;
            _state := Pusher_states_t#First_Slide_Timer_Metal;
        END_IF;
        {* end(transition) *}
        {* begin(onExit) *}
        {* end(onExit) *}
        {* end(State) *}

    Pusher_states_t#First_Slide_white_workpieces:
        {* begin(State) *}
        {* begin(onEntry) *}
        _transit := FALSE;
        {* end(onEntry) *}
        {* begin(onActive) *}
        {* end(onActive) *}
        {* begin(transition) *}
        IF TRUE THEN
            _transit := TRUE;
            _state := Pusher_states_t#First_Slide_Timer_White;
        END_IF;
        {* end(transition) *}
        {* begin(onExit) *}
        {* end(onExit) *}
        {* end(State) *}

    Pusher_states_t#Init:
        {* begin(State) *}
        {* begin(onEntry) *}
        _transit := FALSE;
        {* end(onEntry) *}
        {* begin(onActive) *}
        {* end(onActive) *}
        {* begin(transition) *}
        IF StartVar THEN
            _transit := TRUE;
            _state := Pusher_states_t#Interstep;
        END_IF;
        {* end(transition) *}
        {* begin(onExit) *}
        {* end(onExit) *}
        {* end(State) *}

    Pusher_states_t#Interstep:
        {* begin(State) *}
        {* begin(onEntry) *}
        _transit := FALSE;
        {* end(onEntry) *}
        {* begin(onActive) *}
        PusherY1 := FALSE;
        PusherY2 := FALSE;
        interconnect2 := FALSE;
        interconnect3 := FALSE;
        StartVar := FALSE;
        interconnect_Slide1_Black := FALSE;
        interconnect_Slide2_Black := FALSE;
        interconnect_Slide1_White := FALSE;
        interconnect_Slide2_White := FALSE;
        interconnect_Slide1_Metal := FALSE;
        interconnect_Slide2_Metal := FALSE;
        {* end(onActive) *}
        {* begin(transition) *}
        IF TRUE THEN
            _transit := TRUE;
            _state := Pusher_states_t#Interstep_2;
        END_IF;
        {* end(transition) *}
        {* begin(onExit) *}
        {* end(onExit) *}
        {* end(State) *}

    Pusher_states_t#Interstep_2:
        {* begin(State) *}
        {* begin(onEntry) *}
        _transit := FALSE;
        {* end(onEntry) *}
        {* begin(onActive) *}
        {* end(onActive) *}
        {* begin(transition) *}
        IF ((SorterLightnessSensorPusher1 AND SorterCapacitiveSensorPusher1) AND (Priority_Var_Metal > INT#0)) THEN
            _transit := TRUE;
            _state := Pusher_states_t#Check_For_Metal;
        ELSEIF ((NOT SorterLightnesssensorCraneInterfaceInverse AND SorterLightbarrierCraneInterface) AND (Priority_Var_Black > INT#0)) THEN
            _transit := TRUE;
            _state := Pusher_states_t#Check_For_Black;
        ELSEIF ((SorterLightnessSensorPusher1 AND NOT SorterCapacitiveSensorPusher1) AND (Priority_Var_White > INT#0)) THEN
            _transit := TRUE;
            _state := Pusher_states_t#Check_For_White;
        END_IF;
        {* end(transition) *}
        {* begin(onExit) *}
        {* end(onExit) *}
        {* end(State) *}

    Pusher_states_t#PusherY1_Move_In_Black:
        {* begin(State) *}
        {* begin(onEntry) *}
        _transit := FALSE;
        {* end(onEntry) *}
        {* begin(onActive) *}
        IF ((SorterPusher1MovedOut = TRUE) AND (SorterPusher1MovedIn = FALSE)) THEN
            PusherY1 := FALSE;
        END_IF;
        {* end(onActive) *}
        {* begin(transition) *}
        IF SorterPusher1MovedIn THEN
            _transit := TRUE;
            _state := Pusher_states_t#Reset_interconnect_Slide1_Black;
        END_IF;
        {* end(transition) *}
        {* begin(onExit) *}
        {* end(onExit) *}
        {* end(State) *}

    Pusher_states_t#PusherY1_Move_In_Metal:
        {* begin(State) *}
        {* begin(onEntry) *}
        _transit := FALSE;
        {* end(onEntry) *}
        {* begin(onActive) *}
        IF ((SorterPusher1MovedOut = TRUE) AND (SorterPusher1MovedIn = FALSE)) THEN
            PusherY1 := FALSE;
        END_IF;
        {* end(onActive) *}
        {* begin(transition) *}
        IF SorterPusher1MovedIn THEN
            _transit := TRUE;
            _state := Pusher_states_t#Reset_interconnect_Slide1_Metal;
        END_IF;
        {* end(transition) *}
        {* begin(onExit) *}
        {* end(onExit) *}
        {* end(State) *}

    Pusher_states_t#PusherY1_Move_In_White:
        {* begin(State) *}
        {* begin(onEntry) *}
        _transit := FALSE;
        {* end(onEntry) *}
        {* begin(onActive) *}
        IF ((SorterPusher1MovedOut = TRUE) AND (SorterPusher1MovedIn = FALSE)) THEN
            PusherY1 := FALSE;
        END_IF;
        {* end(onActive) *}
        {* begin(transition) *}
        IF SorterPusher1MovedIn THEN
            _transit := TRUE;
            _state := Pusher_states_t#Reset_interconnect_Slide1_White;
        END_IF;
        {* end(transition) *}
        {* begin(onExit) *}
        {* end(onExit) *}
        {* end(State) *}

    Pusher_states_t#PusherY1_Move_Out_Black:
        {* begin(State) *}
        {* begin(onEntry) *}
        _transit := FALSE;
        {* end(onEntry) *}
        {* begin(onActive) *}
        IF ((SorterPusher1MovedOut = FALSE) AND (SorterPusher1MovedIn = TRUE)) THEN
            PusherY1 := TRUE;
        END_IF;
        {* end(onActive) *}
        {* begin(transition) *}
        IF SorterPusher1MovedOut THEN
            _transit := TRUE;
            _state := Pusher_states_t#Wait_Y1_Black;
        END_IF;
        {* end(transition) *}
        {* begin(onExit) *}
        {* end(onExit) *}
        {* end(State) *}

    Pusher_states_t#PusherY1_Move_Out_Metal:
        {* begin(State) *}
        {* begin(onEntry) *}
        _transit := FALSE;
        {* end(onEntry) *}
        {* begin(onActive) *}
        IF ((SorterPusher1MovedOut = FALSE) AND (SorterPusher1MovedIn = TRUE)) THEN
            PusherY1 := TRUE;
        END_IF;
        {* end(onActive) *}
        {* begin(transition) *}
        IF SorterPusher1MovedOut THEN
            _transit := TRUE;
            _state := Pusher_states_t#Wait_Y1_Metal;
        END_IF;
        {* end(transition) *}
        {* begin(onExit) *}
        {* end(onExit) *}
        {* end(State) *}
